KUKA KRL program: EPS_2_25694_GD06_A_20260114065907.src

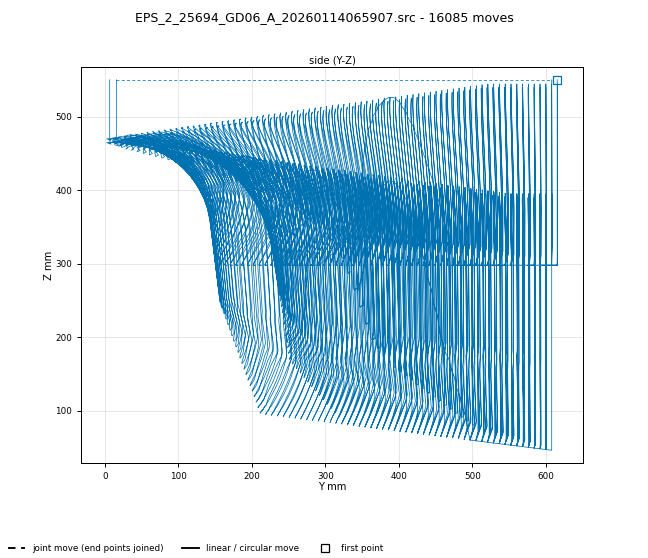
[picture p0: tool path of EPS_2_25694_GD06_A_20260114065907.src, 16085 of 16087 moves have a stored position in this frame; points joined in program order, loops and branches not executed]
&ACCESS RVP
&REL 4
&COMMENT QRS 19112012
&PARAM EDITMASK = *
DEF PART()
EXT BAS (BAS_COMMAND :IN,REAL :IN )
INT I
BAS (#INITMOV,0 )

;KUKA QRS Post kuka4.cps  Date:22-06-2017 !

File_ID=2966

QRS_PRE_INIT()

;Init var - Until changes are made in qrs_pre_init
Outlet_Square_prg=0
Inlet_1_Square_prg=0
Inlet_2_Square_prg=0
Inlet_3_Square_prg=0
Inlet_4_Square_prg=0
Inlet_5_Square_prg=0

Outlet_1={X 0.000, Y 524.050, Z 357.000, B 0.000, E1 0.000 }
Inlet_1={X 0.000, Y 548.960, Z 269.500, B 0.000, E1 174.000 }
Inlet_2={X 0.000, Y 548.960, Z 269.500, B 0.000, E1 220.000 }
Outlet_1_type=366
Inlet_1_type=201
Inlet_2_type=201
;QRS#1=Sidecore dimensions
;QRS#2=375-15" PVC SDR 35
;QRS#3=200-8" PVC SDR 35
;QRS#4=200-8" PVC SDR 35
;QRS#5=
;QRS#6=
;QRS#7=
;QRS#8=
;QRS#9=20Y PSX
;QRS#10=12-08 PSX
;QRS#11=12-08 PSX
;QRS#12=
;QRS#13=
;QRS#14=
;QRS#15=
;QRS#16=1220x127x838 2,75'
;QRS#17=EPS Height
;QRS#18=540
;QRS#19=*
;QRS#20= UPDATED VERSION 22-06-2017
;QRS#21=*
Outlet_Square=0250
Inlet_1_Square=0100
Inlet_2_Square=0100
Inlet_3_Square=0
Inlet_4_Square=0
Inlet_5_Square=0
Mill_Square=1
Outlet_Square_Prg=252
Inlet_1_Square_prg=204
Inlet_2_Square_prg=204

QRS_INIT()

$ADVANCE=5

; T1
PTP {E1 172.623,E2 172.623}
PTP {X 0,Y 615.402,A -85,B 0,C 180,E1 172.623,E2 172.623,E3 0,E4 0,E5 0,E6 0}
QRS_SPEED_INIT()
LIN {X 0,Y 615.402,Z 550,A -85,B 0,C 180,E1 172.623,E2 172.623,E3 0,E4 0,E5 0,E6 0} C_VEL
LIN {X 0,Y 615.402,Z 299.81,A -85,B 0,C 180,E1 172.623,E2 172.623} C_VEL
LIN {X 0,Y 615.427,Z 297.81,A -85,B 0,C 180,E1 172.809,E2 172.809} C_VEL
LIN {X 0,Y 615.817,Z 297.81,A -85,B 0,C 180,E1 174.193,E2 174.193} C_VEL
LIN {X 0,Y 615.867,Z 297.81,A -85,B 0,C 180,E1 178.841,E2 178.841} C_VEL
LIN {X 0,Y 615.867,Z 297.81,A -85,B 0,C 180,E1 183.48,E2 183.48} C_VEL
LIN {X 0,Y 615.824,Z 297.81,A -85,B 0,C 180,E1 188.143,E2 188.143} C_VEL
LIN {X 0,Y 615.832,Z 297.81,A -85,B 0,C 180,E1 192.861,E2 192.861} C_VEL
LIN {X 0,Y 615.792,Z 297.81,A -85,B 0,C 180,E1 197.671,E2 197.671} C_VEL
LIN {X 0,Y 615.792,Z 297.81,A -85,B 0,C 180,E1 197.997,E2 197.997} C_VEL
LIN {X 0,Y 615.78,Z 297.81,A -85,B 0,C 180,E1 202.613,E2 202.613} C_VEL
LIN {X 0,Y 615.256,Z 297.81,A -85,B 0,C 180,E1 205.172,E2 205.172} C_VEL
LIN {X 0,Y 615.748,Z 297.81,A -85,B 0,C 180,E1 207.741,E2 207.741} C_VEL
LIN {X 0,Y 615.184,Z 297.81,A -85,B 0,C 180,E1 210.425,E2 210.425} C_VEL
LIN {X 0,Y 615.704,Z 297.81,A -85,B 0,C 180,E1 213.124,E2 213.124} C_VEL
LIN {X 0,Y 615.631,Z 297.81,A -85,B 0,C 180,E1 213.914,E2 213.914} C_VEL
LIN {X 0,Y 615.66,Z 297.81,A -85,B 0,C 180,E1 218.863,E2 218.863} C_VEL
LIN {X 0,Y 615.262,Z 297.81,A -85,B 0,C 180,E1 221.942,E2 221.942} C_VEL
LIN {X 0,Y 615.675,Z 297.81,A -85,B 0,C 180,E1 224.897,E2 224.897} C_VEL
LIN {X 0,Y 615.638,Z 297.81,A -85,B 0,C 180,E1 228.498,E2 228.498} C_VEL
LIN {X 0,Y 615.376,Z 297.81,A -85,B 0,C 180,E1 231.118,E2 231.118} C_VEL
LIN {X 0,Y 615.432,Z 297.81,A -85,B 0,C 180,E1 232.156,E2 232.156} C_VEL
LIN {X 0,Y 615.702,Z 297.81,A -85,B 0,C 180,E1 234.062,E2 234.062} C_VEL
LIN {X 0,Y 615.153,Z 297.81,A -85,B 0,C 180,E1 236.844,E2 236.844} C_VEL
LIN {X 0,Y 615.737,Z 297.81,A -85,B 0,C 180,E1 239.607,E2 239.607} C_VEL
LIN {X 0,Y 615.234,Z 297.81,A -85,B 0,C 180,E1 242.236,E2 242.236} C_VEL
LIN {X 0,Y 615.794,Z 297.81,A -85,B 0,C 180,E1 244.853,E2 244.853} C_VEL
LIN {X 0,Y 615.734,Z 297.81,A -85,B 0,C 180,E1 247.988,E2 247.988} C_VEL
LIN {X 0,Y 615.838,Z 297.81,A -85,B 0,C 180,E1 248.694,E2 248.694} C_VEL
LIN {X 0,Y 615.498,Z 297.81,A -85,B 0,C 180,E1 249.163,E2 249.163} C_VEL
LIN {X 0,Y 615.621,Z 310.955,A -85,B 0,C 180,E1 249.342,E2 249.342} C_VEL
LIN {X 0,Y 615.725,Z 356.141,A -85,B 0,C 180,E1 249.896,E2 249.896} C_VEL
LIN {X 0,Y 615.805,Z 368.255,A -85,B 0,C 180,E1 250.073,E2 250.073} C_VEL
LIN {X 0,Y 615.746,Z 379.719,A -85,B 0,C 180,E1 250.302,E2 250.302} C_VEL
LIN {X 0,Y 615.701,Z 387.593,A -85,B 0,C 180,E1 250.493,E2 250.493} C_VEL
LIN {X 0,Y 615.787,Z 397.991,A -85,B 0,C 180,E1 250.803,E2 250.803} C_VEL
LIN {X 0,Y 615.773,Z 406.896,A -85,B 0,C 180,E1 251.109,E2 251.109} C_VEL
LIN {X 0,Y 615.749,Z 416.189,A -85,B 0,C 180,E1 251.476,E2 251.476} C_VEL
LIN {X 0,Y 615.792,Z 425.493,A -85,B 0,C 180,E1 251.897,E2 251.897} C_VEL
LIN {X 0,Y 615.792,Z 434.075,A -85,B 0,C 180,E1 252.331,E2 252.331} C_VEL
LIN {X 0,Y 615.784,Z 442.97,A -85,B 0,C 180,E1 252.832,E2 252.832} C_VEL
LIN {X 0,Y 615.789,Z 450.993,A -85,B 0,C 180,E1 253.333,E2 253.333} C_VEL
LIN {X 0,Y 615.781,Z 459.321,A -85,B 0,C 180,E1 253.906,E2 253.906} C_VEL
LIN {X 0,Y 615.8,Z 466.259,A -85,B 0,C 180,E1 254.428,E2 254.428} C_VEL
LIN {X 0,Y 615.798,Z 473.812,A -85,B 0,C 180,E1 255.049,E2 255.049} C_VEL
LIN {X 0,Y 615.765,Z 480.491,A -85,B 0,C 180,E1 255.648,E2 255.648} C_VEL
LIN {X 0,Y 615.798,Z 486.621,A -85,B 0,C 180,E1 256.246,E2 256.246} C_VEL
LIN {X 0,Y 615.819,Z 492.276,A -85,B 0,C 180,E1 256.842,E2 256.842} C_VEL
LIN {X 0,Y 615.737,Z 498.725,A -85,B 0,C 180,E1 257.584,E2 257.584} C_VEL
LIN {X 0,Y 615.725,Z 504.582,A -85,B 0,C 180,E1 258.325,E2 258.325} C_VEL
LIN {X 0,Y 615.783,Z 508.909,A -85,B 0,C 180,E1 258.917,E2 258.917} C_VEL
LIN {X 0,Y 615.79,Z 514.734,A -85,B 0,C 180,E1 259.802,E2 259.802} C_VEL
LIN {X 0,Y 615.671,Z 519.943,A -85,B 0,C 180,E1 260.683,E2 260.683} C_VEL
LIN {X 0,Y 615.681,Z 523.126,A -85,B 0,C 180,E1 261.27,E2 261.27} C_VEL
LIN {X 0,Y 615.809,Z 527.25,A -85,B 0,C 180,E1 262.129,E2 262.129} C_VEL
LIN {X 0,Y 615.715,Z 531.738,A -85,B 0,C 180,E1 263.207,E2 263.207} C_VEL
LIN {X 0,Y 615.679,Z 534.167,A -85,B 0,C 180,E1 263.864,E2 263.864} C_VEL
LIN {X 0,Y 615.737,Z 536.697,A -85,B 0,C 180,E1 264.659,E2 264.659} C_VEL
LIN {X 0,Y 615.8,Z 539.18,A -85,B 0,C 180,E1 265.591,E2 265.591} C_VEL
LIN {X 0,Y 615.655,Z 541.197,A -85,B 0,C 180,E1 266.52,E2 266.52} C_VEL
LIN {X 0,Y 615.667,Z 542.698,A -85,B 0,C 180,E1 267.449,E2 267.449} C_VEL
LIN {X 0,Y 615.73,Z 543.233,A -85,B 0,C 180,E1 267.913,E2 267.913} C_VEL
LIN {X 0,Y 615.79,Z 544.034,A -85,B 0,C 180,E1 268.841,E2 268.841} C_VEL
LIN {X 0,Y 615.643,Z 544.415,A -85,B 0,C 180,E1 269.769,E2 269.769} C_VEL
LIN {X 0,Y 615.659,Z 544.303,A -85,B 0,C 180,E1 270.697,E2 270.697} C_VEL
LIN {X 0,Y 615.728,Z 544.045,A -85,B 0,C 180,E1 271.16,E2 271.16} C_VEL
LIN {X 0,Y 615.709,Z 542.688,A -85,B 0,C 180,E1 272.553,E2 272.553} C_VEL
LIN {X 0,Y 615.632,Z 541.198,A -85,B 0,C 180,E1 273.482,E2 273.482} C_VEL
LIN {X 0,Y 615.743,Z 539.186,A -85,B 0,C 180,E1 274.411,E2 274.411} C_VEL
LIN {X 0,Y 615.793,Z 536.681,A -85,B 0,C 180,E1 275.342,E2 275.342} C_VEL
LIN {X 0,Y 615.685,Z 533.647,A -85,B 0,C 180,E1 276.284,E2 276.284} C_VEL
LIN {X 0,Y 615.732,Z 530.365,A -85,B 0,C 180,E1 277.148,E2 277.148} C_VEL
LIN {X 0,Y 615.811,Z 525.949,A -85,B 0,C 180,E1 278.144,E2 278.144} C_VEL
LIN {X 0,Y 615.693,Z 521.532,A -85,B 0,C 180,E1 279.025,E2 279.025} C_VEL
LIN {X 0,Y 615.673,Z 518.31,A -85,B 0,C 180,E1 279.613,E2 279.613} C_VEL
LIN {X 0,Y 615.794,Z 512.856,A -85,B 0,C 180,E1 280.494,E2 280.494} C_VEL
LIN {X 0,Y 615.803,Z 507.842,A -85,B 0,C 180,E1 281.232,E2 281.232} C_VEL
LIN {X 0,Y 615.711,Z 501.118,A -85,B 0,C 180,E1 282.122,E2 282.122} C_VEL
LIN {X 0,Y 615.758,Z 494.899,A -85,B 0,C 180,E1 282.863,E2 282.863} C_VEL
LIN {X 0,Y 615.835,Z 489.481,A -85,B 0,C 180,E1 283.457,E2 283.457} C_VEL
LIN {X 0,Y 615.797,Z 483.617,A -85,B 0,C 180,E1 284.054,E2 284.054} C_VEL
LIN {X 0,Y 615.767,Z 477.229,A -85,B 0,C 180,E1 284.654,E2 284.654} C_VEL
LIN {X 0,Y 615.775,Z 469.18,A -85,B 0,C 180,E1 285.339,E2 285.339} C_VEL
LIN {X 0,Y 615.798,Z 462.064,A -85,B 0,C 180,E1 285.893,E2 285.893} C_VEL
LIN {X 0,Y 615.802,Z 454.236,A -85,B 0,C 180,E1 286.45,E2 286.45} C_VEL
LIN {X 0,Y 615.788,Z 445.662,A -85,B 0,C 180,E1 287.005,E2 287.005} C_VEL
LIN {X 0,Y 615.783,Z 437.089,A -85,B 0,C 180,E1 287.505,E2 287.505} C_VEL
LIN {X 0,Y 615.774,Z 429.098,A -85,B 0,C 180,E1 287.926,E2 287.926} C_VEL
LIN {X 0,Y 615.807,Z 420.867,A -85,B 0,C 180,E1 288.317,E2 288.317} C_VEL
LIN {X 0,Y 615.769,Z 412.278,A -85,B 0,C 180,E1 288.684,E2 288.684} C_VEL
LIN {X 0,Y 615.728,Z 403.668,A -85,B 0,C 180,E1 289.009,E2 289.009} C_VEL
LIN {X 0,Y 615.82,Z 392.91,A -85,B 0,C 180,E1 289.352,E2 289.352} C_VEL
LIN {X 0,Y 615.806,Z 383.689,A -85,B 0,C 180,E1 289.602,E2 289.602} C_VEL
LIN {X 0,Y 615.724,Z 374.227,A -85,B 0,C 180,E1 289.816,E2 289.816} C_VEL
LIN {X 0,Y 615.718,Z 364.366,A -85,B 0,C 180,E1 289.99,E2 289.99} C_VEL
LIN {X 0,Y 615.684,Z 340.1,A -85,B 0,C 180,E1 290.3,E2 290.3} C_VEL
LIN {X 0,Y 615.604,Z 309.449,A -85,B 0,C 180,E1 290.677,E2 290.677} C_VEL
LIN {X 0,Y 615.662,Z 297.81,A -85,B 0,C 180,E1 290.924,E2 290.924} C_VEL
LIN {X 0,Y 615.846,Z 297.81,A -85,B 0,C 180,E1 291.275,E2 291.275} C_VEL
LIN {X 0,Y 615.834,Z 297.81,A -85,B 0,C 180,E1 292.611,E2 292.611} C_VEL
LIN {X 0,Y 615.254,Z 297.81,A -85,B 0,C 180,E1 295.172,E2 295.172} C_VEL
LIN {X 0,Y 615.755,Z 297.81,A -85,B 0,C 180,E1 297.741,E2 297.741} C_VEL
LIN {X 0,Y 615.188,Z 297.81,A -85,B 0,C 180,E1 300.425,E2 300.425} C_VEL
LIN {X 0,Y 615.704,Z 297.81,A -85,B 0,C 180,E1 303.125,E2 303.125} C_VEL
LIN {X 0,Y 615.639,Z 297.81,A -85,B 0,C 180,E1 303.912,E2 303.912} C_VEL
LIN {X 0,Y 615.631,Z 297.81,A -85,B 0,C 180,E1 308.865,E2 308.865} C_VEL
LIN {X 0,Y 615.208,Z 297.81,A -85,B 0,C 180,E1 311.946,E2 311.946} C_VEL
LIN {X 0,Y 615.608,Z 297.81,A -85,B 0,C 180,E1 314.888,E2 314.888} C_VEL
LIN {X 0,Y 615.621,Z 297.81,A -85,B 0,C 180,E1 318.5,E2 318.5} C_VEL
LIN {X 0,Y 615.341,Z 297.81,A -85,B 0,C 180,E1 321.113,E2 321.113} C_VEL
LIN {X 0,Y 615.391,Z 297.81,A -85,B 0,C 180,E1 322.16,E2 322.16} C_VEL
LIN {X 0,Y 615.638,Z 297.81,A -85,B 0,C 180,E1 324.056,E2 324.056} C_VEL
LIN {X 0,Y 615.107,Z 297.81,A -85,B 0,C 180,E1 326.839,E2 326.839} C_VEL
LIN {X 0,Y 615.705,Z 297.81,A -85,B 0,C 180,E1 329.604,E2 329.604} C_VEL
LIN {X 0,Y 615.204,Z 297.81,A -85,B 0,C 180,E1 332.233,E2 332.233} C_VEL
LIN {X 0,Y 615.747,Z 297.81,A -85,B 0,C 180,E1 334.85,E2 334.85} C_VEL
LIN {X 0,Y 615.745,Z 297.81,A -85,B 0,C 180,E1 339.877,E2 339.877} C_VEL
LIN {X 0,Y 615.773,Z 297.81,A -85,B 0,C 180,E1 343.783,E2 343.783} C_VEL
LIN {X 0,Y 615.771,Z 297.81,A -85,B 0,C 180,E1 349.506,E2 349.506} C_VEL
LIN {X 0,Y 615.834,Z 297.81,A -85,B 0,C 180,E1 354.193,E2 354.193} C_VEL
LIN {X 0,Y 615.858,Z 297.81,A -85,B 0,C 180,E1 358.841,E2 358.841} C_VEL
LIN {X 0,Y 615.81,Z 297.81,A -85,B 0,C 180,E1 363.48,E2 363.48} C_VEL
LIN {X 0,Y 615.85,Z 297.81,A -85,B 0,C 180,E1 368.143,E2 368.143} C_VEL
LIN {X 0,Y 615.774,Z 297.81,A -85,B 0,C 180,E1 372.862,E2 372.862} C_VEL
LIN {X 0,Y 615.794,Z 297.81,A -85,B 0,C 180,E1 377.671,E2 377.671} C_VEL
LIN {X 0,Y 615.796,Z 297.81,A -85,B 0,C 180,E1 377.992,E2 377.992} C_VEL
LIN {X 0,Y 615.745,Z 297.81,A -85,B 0,C 180,E1 382.614,E2 382.614} C_VEL
LIN {X 0,Y 615.221,Z 297.81,A -85,B 0,C 180,E1 385.173,E2 385.173} C_VEL
LIN {X 0,Y 615.747,Z 297.81,A -85,B 0,C 180,E1 387.741,E2 387.741} C_VEL
LIN {X 0,Y 615.229,Z 297.81,A -85,B 0,C 180,E1 390.422,E2 390.422} C_VEL
LIN {X 0,Y 615.823,Z 297.81,A -85,B 0,C 180,E1 393.117,E2 393.117} C_VEL
LIN {X 0,Y 615.838,Z 297.81,A -85,B 0,C 180,E1 397.92,E2 397.92} C_VEL
LIN {X 0,Y 615.79,Z 297.81,A -85,B 0,C 180,E1 398.066,E2 398.066} C_VEL
LIN {X 0,Y 615.611,Z 297.81,A -85,B 0,C 180,E1 398.128,E2 398.128} C_VEL
LIN {X 0,Y 615.791,Z 307.271,A -85,B 0,C 180,E1 398.409,E2 398.409} C_VEL
LIN {X 0,Y 615.852,Z 316.431,A -85,B 0,C 180,E1 398.75,E2 398.75} C_VEL
LIN {X 0,Y 615.848,Z 324.058,A -85,B 0,C 180,E1 399.093,E2 399.093} C_VEL
LIN {X 0,Y 615.861,Z 331.763,A -85,B 0,C 180,E1 399.5,E2 399.5} C_VEL
LIN {X 0,Y 615.839,Z 338.539,A -85,B 0,C 180,E1 399.916,E2 399.916} C_VEL
LIN {X 0,Y 615.815,Z 346.275,A -85,B 0,C 180,E1 400.463,E2 400.463} C_VEL
LIN {X 0,Y 615.85,Z 353.633,A -85,B 0,C 180,E1 401.07,E2 401.07} C_VEL
LIN {X 0,Y 615.809,Z 360.438,A -85,B 0,C 180,E1 401.723,E2 401.723} C_VEL
LIN {X 0,Y 615.772,Z 365.476,A -85,B 0,C 180,E1 402.271,E2 402.271} C_VEL
LIN {X 0,Y 615.81,Z 371.382,A -85,B 0,C 180,E1 403.019,E2 403.019} C_VEL
LIN {X 0,Y 615.813,Z 376.304,A -85,B 0,C 180,E1 403.741,E2 403.741} C_VEL
LIN {X 0,Y 615.749,Z 379.946,A -85,B 0,C 180,E1 404.36,E2 404.36} C_VEL
LIN {X 0,Y 615.79,Z 383.674,A -85,B 0,C 180,E1 405.095,E2 405.095} C_VEL
LIN {X 0,Y 615.832,Z 386.766,A -85,B 0,C 180,E1 405.836,E2 405.836} C_VEL
LIN {X 0,Y 615.744,Z 389.366,A -85,B 0,C 180,E1 406.585,E2 406.585} C_VEL
LIN {X 0,Y 615.764,Z 391.424,A -85,B 0,C 180,E1 407.348,E2 407.348} C_VEL
LIN {X 0,Y 615.84,Z 392.897,A -85,B 0,C 180,E1 408.106,E2 408.106} C_VEL
LIN {X 0,Y 615.797,Z 393.462,A -85,B 0,C 180,E1 408.481,E2 408.481} C_VEL
LIN {X 0,Y 615.766,Z 394.185,A -85,B 0,C 180,E1 409.228,E2 409.228} C_VEL
LIN {X 0,Y 615.803,Z 394.411,A -85,B 0,C 180,E1 409.833,E2 409.833} C_VEL
LIN {X 0,Y 615.843,Z 394.296,A -85,B 0,C 180,E1 410.496,E2 410.496} C_VEL
LIN {X 0,Y 615.768,Z 393.803,A -85,B 0,C 180,E1 411.145,E2 411.145} C_VEL
LIN {X 0,Y 615.795,Z 392.385,A -85,B 0,C 180,E1 412.112,E2 412.112} C_VEL
LIN {X 0,Y 615.822,Z 390.605,A -85,B 0,C 180,E1 412.881,E2 412.881} C_VEL
LIN {X 0,Y 615.73,Z 388.833,A -85,B 0,C 180,E1 413.492,E2 413.492} C_VEL
LIN {X 0,Y 615.742,Z 385.868,A -85,B 0,C 180,E1 414.312,E2 414.312} C_VEL
LIN {X 0,Y 615.829,Z 382.464,A -85,B 0,C 180,E1 415.062,E2 415.062} C_VEL
LIN {X 0,Y 615.787,Z 378.576,A -85,B 0,C 180,E1 415.797,E2 415.797} C_VEL
LIN {X 0,Y 615.8,Z 374.392,A -85,B 0,C 180,E1 416.462,E2 416.462} C_VEL
LIN {X 0,Y 615.851,Z 369.757,A -85,B 0,C 180,E1 417.108,E2 417.108} C_VEL
LIN {X 0,Y 615.805,Z 363.909,A -85,B 0,C 180,E1 417.813,E2 417.813} C_VEL
LIN {X 0,Y 615.811,Z 358.192,A -85,B 0,C 180,E1 418.416,E2 418.416} C_VEL
LIN {X 0,Y 615.849,Z 351.583,A -85,B 0,C 180,E1 419.016,E2 419.016} C_VEL
LIN {X 0,Y 615.82,Z 344.098,A -85,B 0,C 180,E1 419.609,E2 419.609} C_VEL
LIN {X 0,Y 615.835,Z 336.489,A -85,B 0,C 180,E1 420.127,E2 420.127} C_VEL
LIN {X 0,Y 615.822,Z 329.245,A -85,B 0,C 180,E1 420.55,E2 420.55} C_VEL
LIN {X 0,Y 615.826,Z 321.238,A -85,B 0,C 180,E1 420.952,E2 420.952} C_VEL
LIN {X 0,Y 615.807,Z 313.074,A -85,B 0,C 180,E1 421.295,E2 421.295} C_VEL
LIN {X 0,Y 615.702,Z 305.098,A -85,B 0,C 180,E1 421.573,E2 421.573} C_VEL
LIN {X 0,Y 615.384,Z 297.81,A -85,B 0,C 180,E1 421.796,E2 421.796} C_VEL
LIN {X 0,Y 615.784,Z 297.81,A -85,B 0,C 180,E1 421.916,E2 421.916} C_VEL
LIN {X 0,Y 615.706,Z 297.81,A -85,B 0,C 180,E1 423.559,E2 423.559} C_VEL
LIN {X 0,Y 615.767,Z 297.81,A -85,B 0,C 180,E1 424.85,E2 424.85} C_VEL
LIN {X 0,Y 615.813,Z 297.81,A -85,B 0,C 180,E1 429.878,E2 429.878} C_VEL
LIN {X 0,Y 615.83,Z 297.81,A -85,B 0,C 180,E1 433.784,E2 433.784} C_VEL
LIN {X 0,Y 615.806,Z 297.81,A -85,B 0,C 180,E1 439.506,E2 439.506} C_VEL
LIN {X 0,Y 615.79,Z 297.81,A -85,B 0,C 180,E1 443.78,E2 443.78} C_VEL
LIN {X 0,Y 615.666,Z 297.81,A -85,B 0,C 180,E1 443.985,E2 443.985} C_VEL
LIN {X 0,Y 615.253,Z 297.879,A -85,B 0,C 180,E1 444.123,E2 444.123} C_VEL
LIN {X 0,Y 615.743,Z 300.846,A -85,B 0,C 180,E1 444.213,E2 444.213} C_VEL
LIN {X 0,Y 615.794,Z 309.528,A -85,B 0,C 180,E1 444.483,E2 444.483} C_VEL
LIN {X 0,Y 615.801,Z 318.42,A -85,B 0,C 180,E1 444.833,E2 444.833} C_VEL
LIN {X 0,Y 615.828,Z 327,A -85,B 0,C 180,E1 445.24,E2 445.24} C_VEL
LIN {X 0,Y 615.826,Z 335.255,A -85,B 0,C 180,E1 445.705,E2 445.705} C_VEL
LIN {X 0,Y 615.823,Z 342.281,A -85,B 0,C 180,E1 446.17,E2 446.17} C_VEL
LIN {X 0,Y 615.804,Z 348.47,A -85,B 0,C 180,E1 446.635,E2 446.635} C_VEL
LIN {X 0,Y 615.834,Z 355.228,A -85,B 0,C 180,E1 447.216,E2 447.216} C_VEL
LIN {X 0,Y 615.856,Z 361.136,A -85,B 0,C 180,E1 447.796,E2 447.796} C_VEL
LIN {X 0,Y 615.795,Z 366.34,A -85,B 0,C 180,E1 448.376,E2 448.376} C_VEL
LIN {X 0,Y 615.812,Z 371.777,A -85,B 0,C 180,E1 449.072,E2 449.072} C_VEL
LIN {X 0,Y 615.857,Z 376.452,A -85,B 0,C 180,E1 449.767,E2 449.767} C_VEL
LIN {X 0,Y 615.782,Z 380.502,A -85,B 0,C 180,E1 450.463,E2 450.463} C_VEL
LIN {X 0,Y 615.758,Z 383.975,A -85,B 0,C 180,E1 451.159,E2 451.159} C_VEL
LIN {X 0,Y 615.804,Z 385.958,A -85,B 0,C 180,E1 451.623,E2 451.623} C_VEL
LIN {X 0,Y 615.855,Z 387.697,A -85,B 0,C 180,E1 452.086,E2 452.086} C_VEL
LIN {X 0,Y 615.803,Z 389.243,A -85,B 0,C 180,E1 452.551,E2 452.551} C_VEL
LIN {X 0,Y 615.766,Z 390.58,A -85,B 0,C 180,E1 453.015,E2 453.015} C_VEL
LIN {X 0,Y 615.756,Z 391.711,A -85,B 0,C 180,E1 453.48,E2 453.48} C_VEL
LIN {X 0,Y 615.843,Z 393.368,A -85,B 0,C 180,E1 454.409,E2 454.409} C_VEL
LIN {X 0,Y 615.784,Z 393.924,A -85,B 0,C 180,E1 454.875,E2 454.875} C_VEL
LIN {X 0,Y 615.721,Z 394.421,A -85,B 0,C 180,E1 455.807,E2 455.807} C_VEL
LIN {X 0,Y 615.746,Z 394.374,A -85,B 0,C 180,E1 456.281,E2 456.281} C_VEL
LIN {X 0,Y 615.812,Z 394.124,A -85,B 0,C 180,E1 456.756,E2 456.756} C_VEL
LIN {X 0,Y 615.781,Z 393.339,A -85,B 0,C 180,E1 457.535,E2 457.535} C_VEL
LIN {X 0,Y 615.722,Z 392.338,A -85,B 0,C 180,E1 458.143,E2 458.143} C_VEL
LIN {X 0,Y 615.73,Z 391.031,A -85,B 0,C 180,E1 458.73,E2 458.73} C_VEL
LIN {X 0,Y 615.85,Z 388.436,A -85,B 0,C 180,E1 459.609,E2 459.609} C_VEL
LIN {X 0,Y 615.793,Z 386.312,A -85,B 0,C 180,E1 460.198,E2 460.198} C_VEL
LIN {X 0,Y 615.747,Z 383.81,A -85,B 0,C 180,E1 460.788,E2 460.788} C_VEL
LIN {X 0,Y 615.797,Z 379.255,A -85,B 0,C 180,E1 461.674,E2 461.674} C_VEL
LIN {X 0,Y 615.818,Z 374.709,A -85,B 0,C 180,E1 462.415,E2 462.415} C_VEL
LIN {X 0,Y 615.776,Z 369.397,A -85,B 0,C 180,E1 463.158,E2 463.158} C_VEL
LIN {X 0,Y 615.815,Z 364.439,A -85,B 0,C 180,E1 463.754,E2 463.754} C_VEL
LIN {X 0,Y 615.846,Z 358.824,A -85,B 0,C 180,E1 464.351,E2 464.351} C_VEL
LIN {X 0,Y 615.804,Z 352.362,A -85,B 0,C 180,E1 464.951,E2 464.951} C_VEL
LIN {X 0,Y 615.817,Z 344.84,A -85,B 0,C 180,E1 465.556,E2 465.556} C_VEL
LIN {X 0,Y 615.823,Z 338.349,A -85,B 0,C 180,E1 466.006,E2 466.006} C_VEL
LIN {X 0,Y 615.832,Z 330.956,A -85,B 0,C 180,E1 466.458,E2 466.458} C_VEL
LIN {X 0,Y 615.844,Z 323.163,A -85,B 0,C 180,E1 466.86,E2 466.86} C_VEL
LIN {X 0,Y 615.843,Z 315.191,A -85,B 0,C 180,E1 467.213,E2 467.213} C_VEL
LIN {X 0,Y 615.838,Z 306.773,A -85,B 0,C 180,E1 467.516,E2 467.516} C_VEL
LIN {X 0,Y 615.737,Z 297.81,A -85,B 0,C 180,E1 467.787,E2 467.787} C_VEL
LIN {X 0,Y 615.787,Z 297.81,A -85,B 0,C 180,E1 470.121,E2 470.121} C_VEL
LIN {X 0,Y 615.755,Z 297.81,A -85,B 0,C 180,E1 475.148,E2 475.148} C_VEL
LIN {X 0,Y 615.416,Z 297.81,A -85,B 0,C 180,E1 479.461,E2 479.461} C_VEL
LIN {X 0,Y 615.746,Z 297.81,A -85,B 0,C 180,E1 480.393,E2 480.393} C_VEL
LIN {X 0,Y 615.157,Z 297.81,A -85,B 0,C 180,E1 483.845,E2 483.845} C_VEL
LIN {X 0,Y 615.692,Z 297.81,A -85,B 0,C 180,E1 485.939,E2 485.939} C_VEL
LIN {X 0,Y 615.645,Z 297.81,A -85,B 0,C 180,E1 487.87,E2 487.87} C_VEL
LIN {X 0,Y 615.726,Z 297.81,A -85,B 0,C 180,E1 488.856,E2 488.856} C_VEL
LIN {X 0,Y 615.226,Z 297.81,A -85,B 0,C 180,E1 491.943,E2 491.943} C_VEL
LIN {X 0,Y 615.649,Z 297.81,A -85,B 0,C 180,E1 494.892,E2 494.892} C_VEL
LIN {X 0,Y 615.618,Z 297.81,A -85,B 0,C 180,E1 498.498,E2 498.498} C_VEL
LIN {X 0,Y 615.356,Z 297.81,A -85,B 0,C 180,E1 501.114,E2 501.114} C_VEL
LIN {X 0,Y 615.409,Z 297.81,A -85,B 0,C 180,E1 502.155,E2 502.155} C_VEL
LIN {X 0,Y 615.689,Z 297.81,A -85,B 0,C 180,E1 504.059,E2 504.059} C_VEL
LIN {X 0,Y 615.136,Z 297.81,A -85,B 0,C 180,E1 506.841,E2 506.841} C_VEL
LIN {X 0,Y 615.715,Z 297.81,A -85,B 0,C 180,E1 509.604,E2 509.604} C_VEL
LIN {X 0,Y 615.204,Z 297.81,A -85,B 0,C 180,E1 512.233,E2 512.233} C_VEL
LIN {X 0,Y 615.732,Z 297.81,A -85,B 0,C 180,E1 514.849,E2 514.849} C_VEL
LIN {X 0,Y 615.817,Z 297.81,A -85,B 0,C 180,E1 519.879,E2 519.879} C_VEL
LIN {X 0,Y 615.772,Z 297.81,A -85,B 0,C 180,E1 523.3,E2 523.3} C_VEL
LIN {X 0,Y 615.423,Z 297.81,A -85,B 0,C 180,E1 524.738,E2 524.738} C_VEL
LIN {X 0,Y 615.844,Z 297.81,A -85,B 0,C 180,E1 529.507,E2 529.507} C_VEL
LIN {X 0,Y 615.427,Z 297.81,A -85,B 0,C 180,E1 532.809,E2 532.809} C_VEL
LIN {X 0,Y 612.995,Z 297.81,A -85,B 0,C 180,E1 534.011,E2 534.011} C_VEL
LIN {X 0,Y 607.578,Z 297.81,A -85,B 0,C 180,E1 535.808,E2 535.808} C_VEL
LIN {X 0,Y 607.469,Z 297.81,A -85,B 0,C 180,E1 536.015,E2 536.015} C_VEL
LIN {X 0,Y 607.617,Z 297.81,A -85,B 0,C 180,E1 539.991,E2 539.991} C_VEL
LIN {X 0,Y 607.701,Z 297.81,A -85,B 0,C 180,E1 544.263,E2 544.263} C_VEL
LIN {X 0,Y 607.775,Z 297.81,A -85,B 0,C 180,E1 548.558,E2 548.558} C_VEL
LIN {X 0,Y 607.925,Z 297.81,A -85,B 0,C 180,E1 552.9,E2 552.9} C_VEL
LIN {X 0,Y 607.621,Z 297.81,A -85,B 0,C 180,E1 558.827,E2 558.827} C_VEL
LIN {X 0,Y 607.588,Z 297.81,A -85,B 0,C 180,E1 563.405,E2 563.405} C_VEL
LIN {X 0,Y 607.693,Z 297.81,A -85,B 0,C 180,E1 568.142,E2 568.142} C_VEL
LIN {X 0,Y 607.805,Z 297.81,A -85,B 0,C 180,E1 573.097,E2 573.097} C_VEL
LIN {X 0,Y 607.509,Z 297.81,A -85,B 0,C 180,E1 579.645,E2 579.645} C_VEL
LIN {X 0,Y 607.535,Z 297.81,A -85,B 0,C 180,E1 585.935,E2 585.935} C_VEL
LIN {X 0,Y 607.438,Z 297.81,A -85,B 0,C 180,E1 590.351,E2 590.351} C_VEL
LIN {X 0,Y 607.429,Z 297.81,A -85,B 0,C 180,E1 595.153,E2 595.153} C_VEL
LIN {X 0,Y 607.58,Z 297.81,A -85,B 0,C 180,E1 600.359,E2 600.359} C_VEL
LIN {X 0,Y 607.866,Z 297.81,A -85,B 0,C 180,E1 605.038,E2 605.038} C_VEL
LIN {X 0,Y 607.771,Z 297.81,A -85,B 0,C 180,E1 608.899,E2 608.899} C_VEL
LIN {X 0,Y 608.338,Z 378.776,A -85,B 0,C 180,E1 610.029,E2 610.029} C_VEL
LIN {X 0,Y 608.256,Z 411.502,A -85,B 0,C 180,E1 611.046,E2 611.046} C_VEL
LIN {X 0,Y 608.14,Z 444.064,A -85,B 0,C 180,E1 612.676,E2 612.676} C_VEL
LIN {X 0,Y 608.084,Z 472.977,A -85,B 0,C 180,E1 614.78,E2 614.78} C_VEL
LIN {X 0,Y 607.951,Z 497.622,A -85,B 0,C 180,E1 617.274,E2 617.274} C_VEL
LIN {X 0,Y 607.898,Z 516.906,A -85,B 0,C 180,E1 619.993,E2 619.993} C_VEL
LIN {X 0,Y 607.876,Z 531.186,A -85,B 0,C 180,E1 622.87,E2 622.87} C_VEL
LIN {X 0,Y 607.892,Z 540.101,A -85,B 0,C 180,E1 625.729,E2 625.729} C_VEL
LIN {X 0,Y 607.881,Z 544.419,A -85,B 0,C 180,E1 628.577,E2 628.577} C_VEL
LIN {X 0,Y 607.823,Z 544.419,A -85,B 0,C 180,E1 631.422,E2 631.422} C_VEL
LIN {X 0,Y 607.841,Z 540.103,A -85,B 0,C 180,E1 634.271,E2 634.271} C_VEL
LIN {X 0,Y 607.891,Z 530.086,A -85,B 0,C 180,E1 637.39,E2 637.39} C_VEL
LIN {X 0,Y 607.931,Z 514.736,A -85,B 0,C 180,E1 640.367,E2 640.367} C_VEL
LIN {X 0,Y 607.969,Z 494.45,A -85,B 0,C 180,E1 643.09,E2 643.09} C_VEL
LIN {X 0,Y 608.069,Z 468.731,A -85,B 0,C 180,E1 645.575,E2 645.575} C_VEL
LIN {X 0,Y 608.18,Z 439.431,A -85,B 0,C 180,E1 647.601,E2 647.601} C_VEL
LIN {X 0,Y 608.251,Z 407.802,A -85,B 0,C 180,E1 649.098,E2 649.098} C_VEL
LIN {X 0,Y 608.289,Z 373.526,A -85,B 0,C 180,E1 650.082,E2 650.082} C_VEL
LIN {X 0,Y 607.842,Z 297.81,A -85,B 0,C 180,E1 651.098,E2 651.098} C_VEL
LIN {X 0,Y 607.511,Z 297.81,A -85,B 0,C 180,E1 656.61,E2 656.61} C_VEL
LIN {X 0,Y 607.539,Z 297.81,A -85,B 0,C 180,E1 662.397,E2 662.397} C_VEL
LIN {X 0,Y 607.552,Z 297.81,A -85,B 0,C 180,E1 668.384,E2 668.384} C_VEL
LIN {X 0,Y 607.449,Z 297.81,A -85,B 0,C 180,E1 674.071,E2 674.071} C_VEL
LIN {X 0,Y 607.633,Z 297.81,A -85,B 0,C 180,E1 678.16,E2 678.16} C_VEL
LIN {X 0,Y 607.6,Z 297.81,A -85,B 0,C 180,E1 683.422,E2 683.422} C_VEL
LIN {X 0,Y 607.529,Z 297.81,A -85,B 0,C 180,E1 690.381,E2 690.381} C_VEL
LIN {X 0,Y 607.778,Z 297.81,A -85,B 0,C 180,E1 695.043,E2 695.043} C_VEL
LIN {X 0,Y 607.542,Z 297.81,A -85,B 0,C 180,E1 701.171,E2 701.171} C_VEL
LIN {X 0,Y 607.203,Z 297.81,A -85,B 0,C 180,E1 705.619,E2 705.619} C_VEL
LIN {X 0,Y 607.7,Z 297.81,A -85,B 0,C 180,E1 709.999,E2 709.999} C_VEL
LIN {X 0,Y 607.904,Z 297.81,A -85,B 0,C 180,E1 714.31,E2 714.31} C_VEL
LIN {X 0,Y 607.565,Z 297.81,A -85,B 0,C 180,E1 720.009,E2 720.009} C_VEL
LIN {X 0,Y 607.627,Z 297.81,A -85,B 0,C 180,E1 724.282,E2 724.282} C_VEL
LIN {X 0,Y 607.793,Z 297.81,A -85,B 0,C 180,E1 728.576,E2 728.576} C_VEL
LIN {X 0,Y 607.843,Z 297.81,A -85,B 0,C 180,E1 732.92,E2 732.92} C_VEL
LIN {X 0,Y 607.584,Z 297.81,A -85,B 0,C 180,E1 738.846,E2 738.846} C_VEL
LIN {X 0,Y 607.548,Z 297.81,A -85,B 0,C 180,E1 743.426,E2 743.426} C_VEL
LIN {X 0,Y 607.686,Z 297.81,A -85,B 0,C 180,E1 748.163,E2 748.163} C_VEL
LIN {X 0,Y 607.917,Z 297.81,A -85,B 0,C 180,E1 753.111,E2 753.111} C_VEL
LIN {X 0,Y 607.881,Z 297.869,A -85,B 0,C 180,E1 757.977,E2 757.977} C_VEL
LIN {X 0,Y 608.09,Z 324.763,A -85,B 0,C 180,E1 758.983,E2 758.983} C_VEL
LIN {X 0,Y 608.018,Z 347.922,A -85,B 0,C 180,E1 760.458,E2 760.458} C_VEL
LIN {X 0,Y 607.935,Z 366.539,A -85,B 0,C 180,E1 762.267,E2 762.267} C_VEL
LIN {X 0,Y 607.906,Z 381.719,A -85,B 0,C 180,E1 764.541,E2 764.541} C_VEL
LIN {X 0,Y 607.886,Z 391.02,A -85,B 0,C 180,E1 766.949,E2 766.949} C_VEL
LIN {X 0,Y 607.964,Z 393.551,A -85,B 0,C 180,E1 768.141,E2 768.141} C_VEL
LIN {X 0,Y 607.974,Z 394.922,A -85,B 0,C 180,E1 770.318,E2 770.318} C_VEL
LIN {X 0,Y 607.928,Z 391.925,A -85,B 0,C 180,E1 772.606,E2 772.606} C_VEL
LIN {X 0,Y 607.97,Z 383.474,A -85,B 0,C 180,E1 775.01,E2 775.01} C_VEL
LIN {X 0,Y 608.016,Z 369.234,A -85,B 0,C 180,E1 777.311,E2 777.311} C_VEL
LIN {X 0,Y 608.021,Z 349.649,A -85,B 0,C 180,E1 779.315,E2 779.315} C_VEL
LIN {X 0,Y 608.079,Z 326.178,A -85,B 0,C 180,E1 780.856,E2 780.856} C_VEL
LIN {X 0,Y 607.76,Z 300.878,A -85,B 0,C 180,E1 781.853,E2 781.853} C_VEL
LIN {X 0,Y 607.701,Z 297.81,A -85,B 0,C 180,E1 781.959,E2 781.959} C_VEL
LIN {X 0,Y 607.358,Z 297.81,A -85,B 0,C 180,E1 786.577,E2 786.577} C_VEL
LIN {X 0,Y 607.609,Z 297.81,A -85,B 0,C 180,E1 791.165,E2 791.165} C_VEL
LIN {X 0,Y 607.265,Z 297.81,A -85,B 0,C 180,E1 795.612,E2 795.612} C_VEL
LIN {X 0,Y 607.753,Z 297.81,A -85,B 0,C 180,E1 799.991,E2 799.991} C_VEL
LIN {X 0,Y 607.541,Z 298.465,A -85,B 0,C 180,E1 803.986,E2 803.986} C_VEL
LIN {X 0,Y 608.071,Z 323.644,A -85,B 0,C 180,E1 804.928,E2 804.928} C_VEL
LIN {X 0,Y 608.007,Z 346.615,A -85,B 0,C 180,E1 806.354,E2 806.354} C_VEL
LIN {X 0,Y 607.976,Z 366.175,A -85,B 0,C 180,E1 808.223,E2 808.223} C_VEL
LIN {X 0,Y 607.95,Z 380.712,A -85,B 0,C 180,E1 810.356,E2 810.356} C_VEL
LIN {X 0,Y 607.923,Z 390.743,A -85,B 0,C 180,E1 812.846,E2 812.846} C_VEL
LIN {X 0,Y 607.956,Z 393.765,A -85,B 0,C 180,E1 814.271,E2 814.271} C_VEL
LIN {X 0,Y 607.945,Z 394.691,A -85,B 0,C 180,E1 816.765,E2 816.765} C_VEL
LIN {X 0,Y 607.944,Z 390.125,A -85,B 0,C 180,E1 819.285,E2 819.285} C_VEL
LIN {X 0,Y 607.934,Z 379.279,A -85,B 0,C 180,E1 821.817,E2 821.817} C_VEL
LIN {X 0,Y 608.007,Z 363.38,A -85,B 0,C 180,E1 824.004,E2 824.004} C_VEL
LIN {X 0,Y 608.03,Z 342.745,A -85,B 0,C 180,E1 825.843,E2 825.843} C_VEL
LIN {X 0,Y 608.086,Z 319.29,A -85,B 0,C 180,E1 827.186,E2 827.186} C_VEL
LIN {X 0,Y 607.801,Z 297.81,A -85,B 0,C 180,E1 827.987,E2 827.987} C_VEL
LIN {X 0,Y 607.348,Z 297.81,A -85,B 0,C 180,E1 831.882,E2 831.882} C_VEL
LIN {X 0,Y 607.796,Z 297.81,A -85,B 0,C 180,E1 834.965,E2 834.965} C_VEL
LIN {X 0,Y 607.618,Z 297.81,A -85,B 0,C 180,E1 839.782,E2 839.782} C_VEL
LIN {X 0,Y 607.722,Z 297.81,A -85,B 0,C 180,E1 846.579,E2 846.579} C_VEL
LIN {X 0,Y 607.309,Z 297.81,A -85,B 0,C 180,E1 851.79,E2 851.79} C_VEL
LIN {X 0,Y 607.475,Z 297.81,A -85,B 0,C 180,E1 856.086,E2 856.086} C_VEL
LIN {X 0,Y 607.403,Z 297.81,A -85,B 0,C 180,E1 860.368,E2 860.368} C_VEL
LIN {X 0,Y 607.42,Z 297.81,A -85,B 0,C 180,E1 865.141,E2 865.141} C_VEL
LIN {X 0,Y 607.532,Z 297.81,A -85,B 0,C 180,E1 870.382,E2 870.382} C_VEL
LIN {X 0,Y 607.764,Z 297.81,A -85,B 0,C 180,E1 875.023,E2 875.023} C_VEL
LIN {X 0,Y 607.657,Z 297.81,A -85,B 0,C 180,E1 881.156,E2 881.156} C_VEL
LIN {X 0,Y 607.26,Z 297.81,A -85,B 0,C 180,E1 885.726,E2 885.726} C_VEL
LIN {X 0,Y 607.769,Z 297.81,A -85,B 0,C 180,E1 889.982,E2 889.982} C_VEL
LIN {X 0,Y 607.876,Z 297.81,A -85,B 0,C 180,E1 894.292,E2 894.292} C_VEL
LIN {X 0,Y 607.469,Z 297.81,A -85,B 0,C 180,E1 896.015,E2 896.015} C_VEL
LIN {X 0,Y 603.675,Z 297.81,A -85,B 0,C 180,E1 897.627,E2 897.627} C_VEL
LIN {X 0,Y 599.793,Z 297.81,A -85,B 0,C 180,E1 899.26,E2 899.26} C_VEL
LIN {X 0,Y 599.797,Z 297.81,A -85,B 0,C 180,E1 904.32,E2 904.32} C_VEL
LIN {X 0,Y 599.833,Z 297.81,A -85,B 0,C 180,E1 908.673,E2 908.673} C_VEL
LIN {X 0,Y 599.942,Z 297.81,A -85,B 0,C 180,E1 913.075,E2 913.075} C_VEL
LIN {X 0,Y 599.663,Z 297.81,A -85,B 0,C 180,E1 919.086,E2 919.086} C_VEL
LIN {X 0,Y 599.599,Z 297.81,A -85,B 0,C 180,E1 923.736,E2 923.736} C_VEL
LIN {X 0,Y 599.668,Z 297.81,A -85,B 0,C 180,E1 928.553,E2 928.553} C_VEL
LIN {X 0,Y 599.668,Z 297.81,A -85,B 0,C 180,E1 933.859,E2 933.859} C_VEL
LIN {X 0,Y 599.635,Z 297.81,A -85,B 0,C 180,E1 938.976,E2 938.976} C_VEL
LIN {X 0,Y 599.542,Z 297.81,A -85,B 0,C 180,E1 945.191,E2 945.191} C_VEL
LIN {X 0,Y 599.548,Z 297.81,A -85,B 0,C 180,E1 951.007,E2 951.007} C_VEL
LIN {X 0,Y 599.582,Z 297.81,A -85,B 0,C 180,E1 954.63,E2 954.63} C_VEL
LIN {X 0,Y 599.63,Z 297.81,A -85,B 0,C 180,E1 959.78,E2 959.78} C_VEL
LIN {X 0,Y 599.923,Z 297.81,A -85,B 0,C 180,E1 964.875,E2 964.875} C_VEL
LIN {X 0,Y 599.909,Z 297.81,A -85,B 0,C 180,E1 968.596,E2 968.596} C_VEL
LIN {X 0,Y 600.902,Z 335.691,A -85,B 0,C 180,E1 969.122,E2 969.122} C_VEL
LIN {X 0,Y 600.874,Z 380.906,A -85,B 0,C 180,E1 969.822,E2 969.822} C_VEL
LIN {X 0,Y 600.73,Z 414.949,A -85,B 0,C 180,E1 970.94,E2 970.94} C_VEL
LIN {X 0,Y 600.534,Z 446.068,A -85,B 0,C 180,E1 972.575,E2 972.575} C_VEL
LIN {X 0,Y 600.348,Z 474.286,A -85,B 0,C 180,E1 974.697,E2 974.697} C_VEL
LIN {X 0,Y 600.112,Z 499.089,A -85,B 0,C 180,E1 977.289,E2 977.289} C_VEL
LIN {X 0,Y 600.024,Z 519.061,A -85,B 0,C 180,E1 980.226,E2 980.226} C_VEL
LIN {X 0,Y 599.944,Z 533.192,A -85,B 0,C 180,E1 983.32,E2 983.32} C_VEL
LIN {X 0,Y 599.923,Z 541.631,A -85,B 0,C 180,E1 986.394,E2 986.394} C_VEL
LIN {X 0,Y 599.977,Z 544.42,A -85,B 0,C 180,E1 988.558,E2 988.558} C_VEL
LIN {X 0,Y 599.92,Z 544.42,A -85,B 0,C 180,E1 991.441,E2 991.441} C_VEL
LIN {X 0,Y 599.966,Z 540.103,A -85,B 0,C 180,E1 994.327,E2 994.327} C_VEL
LIN {X 0,Y 600.007,Z 529.67,A -85,B 0,C 180,E1 997.587,E2 997.587} C_VEL
LIN {X 0,Y 600.071,Z 515.136,A -85,B 0,C 180,E1 1000.437,E2 1000.437} C_VEL
LIN {X 0,Y 600.189,Z 494.451,A -85,B 0,C 180,E1 1003.263,E2 1003.263} C_VEL
LIN {X 0,Y 600.362,Z 468.864,A -85,B 0,C 180,E1 1005.769,E2 1005.769} C_VEL
LIN {X 0,Y 600.589,Z 439.435,A -85,B 0,C 180,E1 1007.831,E2 1007.831} C_VEL
LIN {X 0,Y 600.726,Z 406.822,A -85,B 0,C 180,E1 1009.386,E2 1009.386} C_VEL
LIN {X 0,Y 600.876,Z 373.869,A -85,B 0,C 180,E1 1010.334,E2 1010.334} C_VEL
LIN {X 0,Y 599.975,Z 297.81,A -85,B 0,C 180,E1 1011.392,E2 1011.392} C_VEL
LIN {X 0,Y 599.737,Z 297.81,A -85,B 0,C 180,E1 1018.297,E2 1018.297} C_VEL
LIN {X 0,Y 599.666,Z 297.81,A -85,B 0,C 180,E1 1023.872,E2 1023.872} C_VEL
LIN {X 0,Y 599.575,Z 297.81,A -85,B 0,C 180,E1 1028.99,E2 1028.99} C_VEL
LIN {X 0,Y 599.483,Z 297.81,A -85,B 0,C 180,E1 1035.197,E2 1035.197} C_VEL
LIN {X 0,Y 599.505,Z 297.81,A -85,B 0,C 180,E1 1041.014,E2 1041.014} C_VEL
LIN {X 0,Y 599.522,Z 297.81,A -85,B 0,C 180,E1 1044.636,E2 1044.636} C_VEL
LIN {X 0,Y 599.592,Z 297.81,A -85,B 0,C 180,E1 1049.788,E2 1049.788} C_VEL
LIN {X 0,Y 599.837,Z 297.81,A -85,B 0,C 180,E1 1054.909,E2 1054.909} C_VEL
LIN {X 0,Y 599.693,Z 297.81,A -85,B 0,C 180,E1 1060.915,E2 1060.915} C_VEL
LIN {X 0,Y 599.343,Z 297.81,A -85,B 0,C 180,E1 1065.426,E2 1065.426} C_VEL
LIN {X 0,Y 599.76,Z 297.81,A -85,B 0,C 180,E1 1069.865,E2 1069.865} C_VEL
LIN {X 0,Y 599.999,Z 297.81,A -85,B 0,C 180,E1 1074.235,E2 1074.235} C_VEL
LIN {X 0,Y 599.664,Z 297.81,A -85,B 0,C 180,E1 1080.009,E2 1080.009} C_VEL
LIN {X 0,Y 599.71,Z 297.81,A -85,B 0,C 180,E1 1084.338,E2 1084.338} C_VEL
LIN {X 0,Y 599.845,Z 297.81,A -85,B 0,C 180,E1 1088.691,E2 1088.691} C_VEL
LIN {X 0,Y 599.868,Z 297.81,A -85,B 0,C 180,E1 1093.095,E2 1093.095} C_VEL
LIN {X 0,Y 599.837,Z 297.81,A -85,B 0,C 180,E1 1097.581,E2 1097.581} C_VEL
LIN {X 0,Y 599.565,Z 297.81,A -85,B 0,C 180,E1 1103.757,E2 1103.757} C_VEL
LIN {X 0,Y 599.658,Z 297.81,A -85,B 0,C 180,E1 1108.574,E2 1108.574} C_VEL
LIN {X 0,Y 599.756,Z 297.81,A -85,B 0,C 180,E1 1113.873,E2 1113.873} C_VEL
LIN {X 0,Y 600.005,Z 297.81,A -85,B 0,C 180,E1 1117.799,E2 1117.799} C_VEL
LIN {X 0,Y 600.314,Z 325.6,A -85,B 0,C 180,E1 1118.881,E2 1118.881} C_VEL
LIN {X 0,Y 600.197,Z 349.487,A -85,B 0,C 180,E1 1120.458,E2 1120.458} C_VEL
LIN {X 0,Y 600.078,Z 368.526,A -85,B 0,C 180,E1 1122.413,E2 1122.413} C_VEL
LIN {X 0,Y 600.033,Z 382.151,A -85,B 0,C 180,E1 1124.557,E2 1124.557} C_VEL
LIN {X 0,Y 599.982,Z 390.86,A -85,B 0,C 180,E1 1126.849,E2 1126.849} C_VEL
LIN {X 0,Y 599.994,Z 394.712,A -85,B 0,C 180,E1 1129.164,E2 1129.164} C_VEL
LIN {X 0,Y 599.997,Z 394.276,A -85,B 0,C 180,E1 1131.245,E2 1131.245} C_VEL
LIN {X 0,Y 599.978,Z 389.239,A -85,B 0,C 180,E1 1133.611,E2 1133.611} C_VEL
LIN {X 0,Y 600.065,Z 378.052,A -85,B 0,C 180,E1 1136.103,E2 1136.103} C_VEL
LIN {X 0,Y 600.125,Z 361.637,A -85,B 0,C 180,E1 1138.303,E2 1138.303} C_VEL
LIN {X 0,Y 600.233,Z 340.091,A -85,B 0,C 180,E1 1140.162,E2 1140.162} C_VEL
LIN {X 0,Y 600.314,Z 316.083,A -85,B 0,C 180,E1 1141.472,E2 1141.472} C_VEL
LIN {X 0,Y 599.963,Z 297.81,A -85,B 0,C 180,E1 1142.17,E2 1142.17} C_VEL
LIN {X 0,Y 599.516,Z 297.81,A -85,B 0,C 180,E1 1146.252,E2 1146.252} C_VEL
LIN {X 0,Y 599.766,Z 297.81,A -85,B 0,C 180,E1 1150.909,E2 1150.909} C_VEL
LIN {X 0,Y 599.404,Z 297.81,A -85,B 0,C 180,E1 1155.419,E2 1155.419} C_VEL
LIN {X 0,Y 599.811,Z 297.81,A -85,B 0,C 180,E1 1159.857,E2 1159.857} C_VEL
LIN {X 0,Y 599.728,Z 297.81,A -85,B 0,C 180,E1 1163.801,E2 1163.801} C_VEL
LIN {X 0,Y 600.305,Z 325.238,A -85,B 0,C 180,E1 1164.863,E2 1164.863} C_VEL
LIN {X 0,Y 600.168,Z 348.727,A -85,B 0,C 180,E1 1166.397,E2 1166.397} C_VEL
LIN {X 0,Y 600.099,Z 368.261,A -85,B 0,C 180,E1 1168.379,E2 1168.379} C_VEL
LIN {X 0,Y 600.069,Z 381.137,A -85,B 0,C 180,E1 1170.361,E2 1170.361} C_VEL
LIN {X 0,Y 600.033,Z 390.951,A -85,B 0,C 180,E1 1172.883,E2 1172.883} C_VEL
LIN {X 0,Y 600.072,Z 393.88,A -85,B 0,C 180,E1 1174.327,E2 1174.327} C_VEL
LIN {X 0,Y 599.954,Z 394.966,A -85,B 0,C 180,E1 1175.775,E2 1175.775} C_VEL
LIN {X 0,Y 599.98,Z 393.29,A -85,B 0,C 180,E1 1177.952,E2 1177.952} C_VEL
LIN {X 0,Y 600.032,Z 386.433,A -85,B 0,C 180,E1 1180.399,E2 1180.399} C_VEL
LIN {X 0,Y 600.103,Z 374.232,A -85,B 0,C 180,E1 1182.711,E2 1182.711} C_VEL
LIN {X 0,Y 600.18,Z 356.545,A -85,B 0,C 180,E1 1184.819,E2 1184.819} C_VEL
LIN {X 0,Y 600.248,Z 335.285,A -85,B 0,C 180,E1 1186.478,E2 1186.478} C_VEL
LIN {X 0,Y 600.356,Z 310.343,A -85,B 0,C 180,E1 1187.697,E2 1187.697} C_VEL
LIN {X 0,Y 599.907,Z 297.81,A -85,B 0,C 180,E1 1188.137,E2 1188.137} C_VEL
LIN {X 0,Y 599.503,Z 297.81,A -85,B 0,C 180,E1 1193.75,E2 1193.75} C_VEL
LIN {X 0,Y 599.415,Z 297.81,A -85,B 0,C 180,E1 1198.576,E2 1198.576} C_VEL
LIN {X 0,Y 599.35,Z 297.81,A -85,B 0,C 180,E1 1203.795,E2 1203.795} C_VEL
LIN {X 0,Y 599.814,Z 297.81,A -85,B 0,C 180,E1 1208.733,E2 1208.733} C_VEL
LIN {X 0,Y 599.512,Z 297.81,A -85,B 0,C 180,E1 1215.174,E2 1215.174} C_VEL
LIN {X 0,Y 599.527,Z 297.81,A -85,B 0,C 180,E1 1220.993,E2 1220.993} C_VEL
LIN {X 0,Y 599.555,Z 297.81,A -85,B 0,C 180,E1 1224.616,E2 1224.616} C_VEL
LIN {X 0,Y 599.599,Z 297.81,A -85,B 0,C 180,E1 1229.768,E2 1229.768} C_VEL
LIN {X 0,Y 599.83,Z 297.81,A -85,B 0,C 180,E1 1234.912,E2 1234.912} C_VEL
LIN {X 0,Y 599.797,Z 297.81,A -85,B 0,C 180,E1 1240.899,E2 1240.899} C_VEL
LIN {X 0,Y 599.423,Z 297.81,A -85,B 0,C 180,E1 1245.41,E2 1245.41} C_VEL
LIN {X 0,Y 599.826,Z 297.81,A -85,B 0,C 180,E1 1249.848,E2 1249.848} C_VEL
LIN {X 0,Y 599.979,Z 297.81,A -85,B 0,C 180,E1 1254.217,E2 1254.217} C_VEL
LIN {X 0,Y 599.793,Z 297.81,A -85,B 0,C 180,E1 1259.26,E2 1259.26} C_VEL
LIN {X 0,Y 595.645,Z 297.81,A -85,B 0,C 180,E1 1260.891,E2 1260.891} C_VEL
LIN {X 0,Y 591.835,Z 297.81,A -85,B 0,C 180,E1 1262.544,E2 1262.544} C_VEL
LIN {X 0,Y 591.893,Z 297.81,A -85,B 0,C 180,E1 1268.79,E2 1268.79} C_VEL
LIN {X 0,Y 591.684,Z 297.81,A -85,B 0,C 180,E1 1274.272,E2 1274.272} C_VEL
LIN {X 0,Y 591.724,Z 297.81,A -85,B 0,C 180,E1 1279.352,E2 1279.352} C_VEL
LIN {X 0,Y 591.631,Z 297.81,A -85,B 0,C 180,E1 1284.076,E2 1284.076} C_VEL
LIN {X 0,Y 591.643,Z 297.81,A -85,B 0,C 180,E1 1288.977,E2 1288.977} C_VEL
LIN {X 0,Y 591.719,Z 297.81,A -85,B 0,C 180,E1 1294.118,E2 1294.118} C_VEL
LIN {X 0,Y 591.542,Z 297.81,A -85,B 0,C 180,E1 1300.067,E2 1300.067} C_VEL
LIN {X 0,Y 591.605,Z 297.81,A -85,B 0,C 180,E1 1305.566,E2 1305.566} C_VEL
LIN {X 0,Y 591.589,Z 297.81,A -85,B 0,C 180,E1 1310.38,E2 1310.38} C_VEL
LIN {X 0,Y 591.497,Z 297.81,A -85,B 0,C 180,E1 1315.857,E2 1315.857} C_VEL
LIN {X 0,Y 591.567,Z 297.81,A -85,B 0,C 180,E1 1321.009,E2 1321.009} C_VEL
LIN {X 0,Y 591.867,Z 297.81,A -85,B 0,C 180,E1 1326.594,E2 1326.594} C_VEL
LIN {X 0,Y 592,Z 297.81,A -85,B 0,C 180,E1 1328.295,E2 1328.295} C_VEL
LIN {X 0,Y 593.528,Z 312.319,A -85,B 0,C 180,E1 1328.553,E2 1328.553} C_VEL
LIN {X 0,Y 593.51,Z 378.641,A -85,B 0,C 180,E1 1329.505,E2 1329.505} C_VEL
LIN {X 0,Y 593.225,Z 411.48,A -85,B 0,C 180,E1 1330.546,E2 1330.546} C_VEL
LIN {X 0,Y 592.925,Z 444.072,A -85,B 0,C 180,E1 1332.217,E2 1332.217} C_VEL
LIN {X 0,Y 592.604,Z 473.242,A -85,B 0,C 180,E1 1334.397,E2 1334.397} C_VEL
LIN {X 0,Y 592.345,Z 497.624,A -85,B 0,C 180,E1 1336.933,E2 1336.933} C_VEL
LIN {X 0,Y 592.176,Z 517.993,A -85,B 0,C 180,E1 1339.91,E2 1339.91} C_VEL
LIN {X 0,Y 592.079,Z 532.289,A -85,B 0,C 180,E1 1342.981,E2 1342.981} C_VEL
LIN {X 0,Y 592.105,Z 540.102,A -85,B 0,C 180,E1 1345.615,E2 1345.615} C_VEL
LIN {X 0,Y 592.073,Z 544.42,A -85,B 0,C 180,E1 1348.539,E2 1348.539} C_VEL
LIN {X 0,Y 592.018,Z 544.421,A -85,B 0,C 180,E1 1351.46,E2 1351.46} C_VEL
LIN {X 0,Y 592.066,Z 540.104,A -85,B 0,C 180,E1 1354.385,E2 1354.385} C_VEL
LIN {X 0,Y 592.151,Z 529.67,A -85,B 0,C 180,E1 1357.688,E2 1357.688} C_VEL
LIN {X 0,Y 592.232,Z 513.781,A -85,B 0,C 180,E1 1360.803,E2 1360.803} C_VEL
LIN {X 0,Y 592.443,Z 493.173,A -85,B 0,C 180,E1 1363.589,E2 1363.589} C_VEL
LIN {X 0,Y 592.662,Z 467.729,A -85,B 0,C 180,E1 1366.074,E2 1366.074} C_VEL
LIN {X 0,Y 593.005,Z 437.758,A -85,B 0,C 180,E1 1368.163,E2 1368.163} C_VEL
LIN {X 0,Y 593.256,Z 406.292,A -85,B 0,C 180,E1 1369.661,E2 1369.661} C_VEL
LIN {X 0,Y 593.497,Z 372.089,A -85,B 0,C 180,E1 1370.634,E2 1370.634} C_VEL
LIN {X 0,Y 592.843,Z 301.233,A -85,B 0,C 180,E1 1371.614,E2 1371.614} C_VEL
LIN {X 0,Y 592.055,Z 297.81,A -85,B 0,C 180,E1 1371.721,E2 1371.721} C_VEL
LIN {X 0,Y 591.737,Z 297.81,A -85,B 0,C 180,E1 1377.323,E2 1377.323} C_VEL
LIN {X 0,Y 591.715,Z 297.81,A -85,B 0,C 180,E1 1384.128,E2 1384.128} C_VEL
LIN {X 0,Y 591.5,Z 297.81,A -85,B 0,C 180,E1 1390.075,E2 1390.075} C_VEL
LIN {X 0,Y 591.546,Z 297.81,A -85,B 0,C 180,E1 1395.582,E2 1395.582} C_VEL
LIN {X 0,Y 591.549,Z 297.81,A -85,B 0,C 180,E1 1400.387,E2 1400.387} C_VEL
LIN {X 0,Y 591.45,Z 297.81,A -85,B 0,C 180,E1 1405.864,E2 1405.864} C_VEL
LIN {X 0,Y 591.545,Z 297.81,A -85,B 0,C 180,E1 1411.018,E2 1411.018} C_VEL
LIN {X 0,Y 591.643,Z 297.81,A -85,B 0,C 180,E1 1415.925,E2 1415.925} C_VEL
LIN {X 0,Y 591.777,Z 297.81,A -85,B 0,C 180,E1 1420.65,E2 1420.65} C_VEL
LIN {X 0,Y 591.481,Z 297.81,A -85,B 0,C 180,E1 1425.228,E2 1425.228} C_VEL
LIN {X 0,Y 591.833,Z 297.81,A -85,B 0,C 180,E1 1429.728,E2 1429.728} C_VEL
LIN {X 0,Y 592.062,Z 297.81,A -85,B 0,C 180,E1 1434.158,E2 1434.158} C_VEL
LIN {X 0,Y 591.764,Z 297.81,A -85,B 0,C 180,E1 1440.009,E2 1440.009} C_VEL
LIN {X 0,Y 591.794,Z 297.81,A -85,B 0,C 180,E1 1444.396,E2 1444.396} C_VEL
LIN {X 0,Y 591.901,Z 297.81,A -85,B 0,C 180,E1 1448.808,E2 1448.808} C_VEL
LIN {X 0,Y 591.661,Z 297.81,A -85,B 0,C 180,E1 1454.267,E2 1454.267} C_VEL
LIN {X 0,Y 591.696,Z 297.81,A -85,B 0,C 180,E1 1459.372,E2 1459.372} C_VEL
LIN {X 0,Y 591.614,Z 297.81,A -85,B 0,C 180,E1 1464.097,E2 1464.097} C_VEL
LIN {X 0,Y 591.644,Z 297.81,A -85,B 0,C 180,E1 1468.998,E2 1468.998} C_VEL
LIN {X 0,Y 591.813,Z 297.81,A -85,B 0,C 180,E1 1474.134,E2 1474.134} C_VEL
LIN {X 0,Y 592.08,Z 298.561,A -85,B 0,C 180,E1 1477.671,E2 1477.671} C_VEL
LIN {X 0,Y 592.581,Z 324.166,A -85,B 0,C 180,E1 1478.662,E2 1478.662} C_VEL
LIN {X 0,Y 592.345,Z 347.389,A -85,B 0,C 180,E1 1480.161,E2 1480.161} C_VEL
LIN {X 0,Y 592.221,Z 367.2,A -85,B 0,C 180,E1 1482.144,E2 1482.144} C_VEL
LIN {X 0,Y 592.15,Z 382.116,A -85,B 0,C 180,E1 1484.477,E2 1484.477} C_VEL
LIN {X 0,Y 592.109,Z 391.68,A -85,B 0,C 180,E1 1487.124,E2 1487.124} C_VEL
LIN {X 0,Y 592.119,Z 394.11,A -85,B 0,C 180,E1 1488.502,E2 1488.502} C_VEL
LIN {X 0,Y 592.041,Z 394.901,A -85,B 0,C 180,E1 1490.417,E2 1490.417} C_VEL
LIN {X 0,Y 592.125,Z 391,A -85,B 0,C 180,E1 1493.049,E2 1493.049} C_VEL
LIN {X 0,Y 592.171,Z 381.324,A -85,B 0,C 180,E1 1495.588,E2 1495.588} C_VEL
LIN {X 0,Y 592.263,Z 366.664,A -85,B 0,C 180,E1 1497.832,E2 1497.832} C_VEL
LIN {X 0,Y 592.385,Z 346.333,A -85,B 0,C 180,E1 1499.834,E2 1499.834} C_VEL
LIN {X 0,Y 592.519,Z 323.038,A -85,B 0,C 180,E1 1501.305,E2 1501.305} C_VEL
LIN {X 0,Y 592.077,Z 297.81,A -85,B 0,C 180,E1 1502.278,E2 1502.278} C_VEL
LIN {X 0,Y 591.532,Z 297.81,A -85,B 0,C 180,E1 1507.503,E2 1507.503} C_VEL
LIN {X 0,Y 591.818,Z 297.81,A -85,B 0,C 180,E1 1512.184,E2 1512.184} C_VEL
LIN {X 0,Y 591.602,Z 297.81,A -85,B 0,C 180,E1 1518.226,E2 1518.226} C_VEL
LIN {X 0,Y 591.896,Z 297.81,A -85,B 0,C 180,E1 1523.645,E2 1523.645} C_VEL
LIN {X 0,Y 592.523,Z 323.186,A -85,B 0,C 180,E1 1524.612,E2 1524.612} C_VEL
LIN {X 0,Y 592.372,Z 346.338,A -85,B 0,C 180,E1 1526.075,E2 1526.075} C_VEL
LIN {X 0,Y 592.289,Z 365.975,A -85,B 0,C 180,E1 1527.993,E2 1527.993} C_VEL
LIN {X 0,Y 592.192,Z 381.549,A -85,B 0,C 180,E1 1530.365,E2 1530.365} C_VEL
LIN {X 0,Y 592.133,Z 391.158,A -85,B 0,C 180,E1 1532.922,E2 1532.922} C_VEL
LIN {X 0,Y 592.16,Z 393.974,A -85,B 0,C 180,E1 1534.385,E2 1534.385} C_VEL
LIN {X 0,Y 592.037,Z 394.961,A -85,B 0,C 180,E1 1536.157,E2 1536.157} C_VEL
LIN {X 0,Y 592.074,Z 391.652,A -85,B 0,C 180,E1 1538.797,E2 1538.797} C_VEL
LIN {X 0,Y 592.112,Z 383.241,A -85,B 0,C 180,E1 1541.196,E2 1541.196} C_VEL
LIN {X 0,Y 592.211,Z 368.814,A -85,B 0,C 180,E1 1543.562,E2 1543.562} C_VEL
LIN {X 0,Y 592.348,Z 349.102,A -85,B 0,C 180,E1 1545.61,E2 1545.61} C_VEL
LIN {X 0,Y 592.531,Z 325.963,A -85,B 0,C 180,E1 1547.157,E2 1547.157} C_VEL
LIN {X 0,Y 592.188,Z 299.413,A -85,B 0,C 180,E1 1548.213,E2 1548.213} C_VEL
LIN {X 0,Y 591.982,Z 297.81,A -85,B 0,C 180,E1 1548.388,E2 1548.388} C_VEL
LIN {X 0,Y 591.669,Z 297.81,A -85,B 0,C 180,E1 1554.084,E2 1554.084} C_VEL
LIN {X 0,Y 591.63,Z 297.81,A -85,B 0,C 180,E1 1559.844,E2 1559.844} C_VEL
LIN {X 0,Y 591.767,Z 297.81,A -85,B 0,C 180,E1 1565.909,E2 1565.909} C_VEL
LIN {X 0,Y 591.596,Z 297.81,A -85,B 0,C 180,E1 1570.057,E2 1570.057} C_VEL
LIN {X 0,Y 591.575,Z 297.81,A -85,B 0,C 180,E1 1575.58,E2 1575.58} C_VEL
LIN {X 0,Y 591.572,Z 297.81,A -85,B 0,C 180,E1 1580.366,E2 1580.366} C_VEL
LIN {X 0,Y 591.642,Z 297.81,A -85,B 0,C 180,E1 1584.704,E2 1584.704} C_VEL
LIN {X 0,Y 591.556,Z 297.81,A -85,B 0,C 180,E1 1590.998,E2 1590.998} C_VEL
LIN {X 0,Y 591.659,Z 297.81,A -85,B 0,C 180,E1 1595.905,E2 1595.905} C_VEL
LIN {X 0,Y 591.875,Z 297.81,A -85,B 0,C 180,E1 1600.634,E2 1600.634} C_VEL
LIN {X 0,Y 591.476,Z 297.81,A -85,B 0,C 180,E1 1605.807,E2 1605.807} C_VEL
LIN {X 0,Y 591.678,Z 297.81,A -85,B 0,C 180,E1 1611.188,E2 1611.188} C_VEL
LIN {X 0,Y 591.718,Z 297.81,A -85,B 0,C 180,E1 1615.603,E2 1615.603} C_VEL
LIN {X 0,Y 591.815,Z 297.81,A -85,B 0,C 180,E1 1619.991,E2 1619.991} C_VEL
LIN {X 0,Y 591.835,Z 297.81,A -85,B 0,C 180,E1 1622.544,E2 1622.544} C_VEL
LIN {X 0,Y 589.399,Z 297.81,A -85,B 0,C 180,E1 1623.794,E2 1623.794} C_VEL
LIN {X 0,Y 583.891,Z 297.81,A -85,B 0,C 180,E1 1625.663,E2 1625.663} C_VEL
LIN {X 0,Y 583.795,Z 297.81,A -85,B 0,C 180,E1 1625.879,E2 1625.879} C_VEL
LIN {X 0,Y 583.753,Z 297.81,A -85,B 0,C 180,E1 1630.795,E2 1630.795} C_VEL
LIN {X 0,Y 583.702,Z 297.81,A -85,B 0,C 180,E1 1634.973,E2 1634.973} C_VEL
LIN {X 0,Y 583.781,Z 297.81,A -85,B 0,C 180,E1 1639.626,E2 1639.626} C_VEL
LIN {X 0,Y 583.678,Z 297.81,A -85,B 0,C 180,E1 1644.425,E2 1644.425} C_VEL
LIN {X 0,Y 583.651,Z 297.81,A -85,B 0,C 180,E1 1649.412,E2 1649.412} C_VEL
LIN {X 0,Y 583.717,Z 297.81,A -85,B 0,C 180,E1 1654.652,E2 1654.652} C_VEL
LIN {X 0,Y 583.609,Z 297.81,A -85,B 0,C 180,E1 1660.261,E2 1660.261} C_VEL
LIN {X 0,Y 583.749,Z 297.81,A -85,B 0,C 180,E1 1666.358,E2 1666.358} C_VEL
LIN {X 0,Y 583.729,Z 297.81,A -85,B 0,C 180,E1 1671.652,E2 1671.652} C_VEL
LIN {X 0,Y 583.571,Z 297.81,A -85,B 0,C 180,E1 1677.11,E2 1677.11} C_VEL
LIN {X 0,Y 583.626,Z 297.81,A -85,B 0,C 180,E1 1682.263,E2 1682.263} C_VEL
LIN {X 0,Y 584.064,Z 297.81,A -85,B 0,C 180,E1 1687.824,E2 1687.824} C_VEL
LIN {X 0,Y 584.073,Z 297.81,A -85,B 0,C 180,E1 1687.989,E2 1687.989} C_VEL
LIN {X 0,Y 586.143,Z 308.497,A -85,B 0,C 180,E1 1688.22,E2 1688.22} C_VEL
LIN {X 0,Y 586.13,Z 377.575,A -85,B 0,C 180,E1 1689.208,E2 1689.208} C_VEL
LIN {X 0,Y 585.754,Z 411.484,A -85,B 0,C 180,E1 1690.287,E2 1690.287} C_VEL
LIN {X 0,Y 585.341,Z 444.076,A -85,B 0,C 180,E1 1691.979,E2 1691.979} C_VEL
LIN {X 0,Y 584.89,Z 473.241,A -85,B 0,C 180,E1 1694.186,E2 1694.186} C_VEL
LIN {X 0,Y 584.577,Z 497.624,A -85,B 0,C 180,E1 1696.756,E2 1696.756} C_VEL
LIN {X 0,Y 584.321,Z 517.993,A -85,B 0,C 180,E1 1699.773,E2 1699.773} C_VEL
LIN {X 0,Y 584.226,Z 531.185,A -85,B 0,C 180,E1 1702.579,E2 1702.579} C_VEL
LIN {X 0,Y 584.202,Z 540.102,A -85,B 0,C 180,E1 1705.555,E2 1705.555} C_VEL
LIN {X 0,Y 584.182,Z 544.421,A -85,B 0,C 180,E1 1708.519,E2 1708.519} C_VEL
LIN {X 0,Y 584.132,Z 544.421,A -85,B 0,C 180,E1 1711.48,E2 1711.48} C_VEL
LIN {X 0,Y 584.17,Z 540.103,A -85,B 0,C 180,E1 1714.444,E2 1714.444} C_VEL
LIN {X 0,Y 584.277,Z 529.67,A -85,B 0,C 180,E1 1717.792,E2 1717.792} C_VEL
LIN {X 0,Y 584.411,Z 513.379,A -85,B 0,C 180,E1 1721.012,E2 1721.012} C_VEL
LIN {X 0,Y 584.673,Z 492.213,A -85,B 0,C 180,E1 1723.888,E2 1723.888} C_VEL
LIN {X 0,Y 584.99,Z 466.588,A -85,B 0,C 180,E1 1726.387,E2 1726.387} C_VEL
LIN {X 0,Y 585.445,Z 437.762,A -85,B 0,C 180,E1 1728.405,E2 1728.405} C_VEL
LIN {X 0,Y 585.788,Z 406.289,A -85,B 0,C 180,E1 1729.922,E2 1729.922} C_VEL
LIN {X 0,Y 586.1,Z 372.899,A -85,B 0,C 180,E1 1730.89,E2 1730.89} C_VEL
LIN {X 0,Y 585.354,Z 302.617,A -85,B 0,C 180,E1 1731.887,E2 1731.887} C_VEL
LIN {X 0,Y 584.094,Z 297.81,A -85,B 0,C 180,E1 1732.078,E2 1732.078} C_VEL
LIN {X 0,Y 583.717,Z 297.81,A -85,B 0,C 180,E1 1738.5,E2 1738.5} C_VEL
LIN {X 0,Y 583.709,Z 297.81,A -85,B 0,C 180,E1 1744.662,E2 1744.662} C_VEL
LIN {X 0,Y 583.566,Z 297.81,A -85,B 0,C 180,E1 1750.274,E2 1750.274} C_VEL
LIN {X 0,Y 583.677,Z 297.81,A -85,B 0,C 180,E1 1756.376,E2 1756.376} C_VEL
LIN {X 0,Y 583.671,Z 297.81,A -85,B 0,C 180,E1 1761.659,E2 1761.659} C_VEL
LIN {X 0,Y 583.521,Z 297.81,A -85,B 0,C 180,E1 1767.117,E2 1767.117} C_VEL
LIN {X 0,Y 583.608,Z 297.81,A -85,B 0,C 180,E1 1772.272,E2 1772.272} C_VEL
LIN {X 0,Y 583.589,Z 297.81,A -85,B 0,C 180,E1 1777.188,E2 1777.188} C_VEL
LIN {X 0,Y 583.843,Z 297.81,A -85,B 0,C 180,E1 1781.941,E2 1781.941} C_VEL
LIN {X 0,Y 583.656,Z 297.81,A -85,B 0,C 180,E1 1788.072,E2 1788.072} C_VEL
LIN {X 0,Y 584.142,Z 297.81,A -85,B 0,C 180,E1 1794.078,E2 1794.078} C_VEL
LIN {X 0,Y 583.886,Z 297.81,A -85,B 0,C 180,E1 1800.009,E2 1800.009} C_VEL
LIN {X 0,Y 583.898,Z 297.81,A -85,B 0,C 180,E1 1804.456,E2 1804.456} C_VEL
LIN {X 0,Y 583.961,Z 297.81,A -85,B 0,C 180,E1 1808.929,E2 1808.929} C_VEL
LIN {X 0,Y 583.966,Z 297.81,A -85,B 0,C 180,E1 1813.458,E2 1813.458} C_VEL
LIN {X 0,Y 583.938,Z 297.81,A -85,B 0,C 180,E1 1818.076,E2 1818.076} C_VEL
LIN {X 0,Y 583.808,Z 297.81,A -85,B 0,C 180,E1 1822.823,E2 1822.823} C_VEL
LIN {X 0,Y 583.721,Z 297.81,A -85,B 0,C 180,E1 1828.486,E2 1828.486} C_VEL
LIN {X 0,Y 583.823,Z 297.81,A -85,B 0,C 180,E1 1834.667,E2 1834.667} C_VEL
LIN {X 0,Y 584.127,Z 298.516,A -85,B 0,C 180,E1 1837.5,E2 1837.5} C_VEL
LIN {X 0,Y 584.827,Z 324.551,A -85,B 0,C 180,E1 1838.53,E2 1838.53} C_VEL
LIN {X 0,Y 584.516,Z 348.064,A -85,B 0,C 180,E1 1840.084,E2 1840.084} C_VEL
LIN {X 0,Y 584.389,Z 366.922,A -85,B 0,C 180,E1 1842.003,E2 1842.003} C_VEL
LIN {X 0,Y 584.264,Z 381.236,A -85,B 0,C 180,E1 1844.228,E2 1844.228} C_VEL
LIN {X 0,Y 584.197,Z 389.666,A -85,B 0,C 180,E1 1846.339,E2 1846.339} C_VEL
LIN {X 0,Y 584.215,Z 394.159,A -85,B 0,C 180,E1 1848.525,E2 1848.525} C_VEL
LIN {X 0,Y 584.122,Z 394.676,A -85,B 0,C 180,E1 1850.823,E2 1850.823} C_VEL
LIN {X 0,Y 584.201,Z 389.723,A -85,B 0,C 180,E1 1853.553,E2 1853.553} C_VEL
LIN {X 0,Y 584.32,Z 379.546,A -85,B 0,C 180,E1 1856.004,E2 1856.004} C_VEL
LIN {X 0,Y 584.394,Z 364.651,A -85,B 0,C 180,E1 1858.183,E2 1858.183} C_VEL
LIN {X 0,Y 584.6,Z 344.067,A -85,B 0,C 180,E1 1860.145,E2 1860.145} C_VEL
LIN {X 0,Y 584.781,Z 320.29,A -85,B 0,C 180,E1 1861.594,E2 1861.594} C_VEL
LIN {X 0,Y 584.164,Z 297.81,A -85,B 0,C 180,E1 1862.43,E2 1862.43} C_VEL
LIN {X 0,Y 583.825,Z 297.81,A -85,B 0,C 180,E1 1868.786,E2 1868.786} C_VEL
LIN {X 0,Y 583.96,Z 297.81,A -85,B 0,C 180,E1 1873.487,E2 1873.487} C_VEL
LIN {X 0,Y 583.935,Z 297.81,A -85,B 0,C 180,E1 1879.579,E2 1879.579} C_VEL
LIN {X 0,Y 584.03,Z 297.81,A -85,B 0,C 180,E1 1883.477,E2 1883.477} C_VEL
LIN {X 0,Y 584.754,Z 322.958,A -85,B 0,C 180,E1 1884.447,E2 1884.447} C_VEL
LIN {X 0,Y 584.552,Z 346.194,A -85,B 0,C 180,E1 1885.93,E2 1885.93} C_VEL
LIN {X 0,Y 584.444,Z 366.632,A -85,B 0,C 180,E1 1887.966,E2 1887.966} C_VEL
LIN {X 0,Y 584.326,Z 381.956,A -85,B 0,C 180,E1 1890.37,E2 1890.37} C_VEL
LIN {X 0,Y 584.251,Z 391.363,A -85,B 0,C 180,E1 1892.961,E2 1892.961} C_VEL
LIN {X 0,Y 584.255,Z 394.066,A -85,B 0,C 180,E1 1894.444,E2 1894.444} C_VEL
LIN {X 0,Y 584.162,Z 394.999,A -85,B 0,C 180,E1 1895.931,E2 1895.931} C_VEL
LIN {X 0,Y 584.179,Z 393.029,A -85,B 0,C 180,E1 1898.168,E2 1898.168} C_VEL
LIN {X 0,Y 584.278,Z 385.686,A -85,B 0,C 180,E1 1900.703,E2 1900.703} C_VEL
LIN {X 0,Y 584.339,Z 373.155,A -85,B 0,C 180,E1 1903.06,E2 1903.06} C_VEL
LIN {X 0,Y 584.461,Z 354.596,A -85,B 0,C 180,E1 1905.25,E2 1905.25} C_VEL
LIN {X 0,Y 584.709,Z 332.442,A -85,B 0,C 180,E1 1906.939,E2 1906.939} C_VEL
LIN {X 0,Y 584.915,Z 307.125,A -85,B 0,C 180,E1 1908.127,E2 1908.127} C_VEL
LIN {X 0,Y 584.096,Z 297.81,A -85,B 0,C 180,E1 1908.433,E2 1908.433} C_VEL
LIN {X 0,Y 583.743,Z 297.81,A -85,B 0,C 180,E1 1914.432,E2 1914.432} C_VEL
LIN {X 0,Y 583.66,Z 297.81,A -85,B 0,C 180,E1 1919.422,E2 1919.422} C_VEL
LIN {X 0,Y 583.639,Z 297.81,A -85,B 0,C 180,E1 1924.668,E2 1924.668} C_VEL
LIN {X 0,Y 583.758,Z 297.81,A -85,B 0,C 180,E1 1929.134,E2 1929.134} C_VEL
LIN {X 0,Y 583.69,Z 297.81,A -85,B 0,C 180,E1 1935.717,E2 1935.717} C_VEL
LIN {X 0,Y 583.709,Z 297.81,A -85,B 0,C 180,E1 1941.638,E2 1941.638} C_VEL
LIN {X 0,Y 583.513,Z 297.81,A -85,B 0,C 180,E1 1947.095,E2 1947.095} C_VEL
LIN {X 0,Y 583.58,Z 297.81,A -85,B 0,C 180,E1 1952.25,E2 1952.25} C_VEL
LIN {X 0,Y 583.627,Z 297.81,A -85,B 0,C 180,E1 1957.17,E2 1957.17} C_VEL
LIN {X 0,Y 583.966,Z 297.81,A -85,B 0,C 180,E1 1961.925,E2 1961.925} C_VEL
LIN {X 0,Y 583.71,Z 297.81,A -85,B 0,C 180,E1 1968.054,E2 1968.054} C_VEL
LIN {X 0,Y 584.132,Z 297.81,A -85,B 0,C 180,E1 1974.059,E2 1974.059} C_VEL
LIN {X 0,Y 583.935,Z 297.81,A -85,B 0,C 180,E1 1979.991,E2 1979.991} C_VEL
LIN {X 0,Y 583.974,Z 297.81,A -85,B 0,C 180,E1 1984.437,E2 1984.437} C_VEL
LIN {X 0,Y 583.795,Z 297.81,A -85,B 0,C 180,E1 1985.879,E2 1985.879} C_VEL
LIN {X 0,Y 579.992,Z 297.81,A -85,B 0,C 180,E1 1987.557,E2 1987.557} C_VEL
LIN {X 0,Y 575.984,Z 297.81,A -85,B 0,C 180,E1 1989.257,E2 1989.257} C_VEL
LIN {X 0,Y 575.937,Z 297.81,A -85,B 0,C 180,E1 1994.203,E2 1994.203} C_VEL
LIN {X 0,Y 575.859,Z 297.81,A -85,B 0,C 180,E1 1999.908,E2 1999.908} C_VEL
LIN {X 0,Y 575.754,Z 297.81,A -85,B 0,C 180,E1 2004.784,E2 2004.784} C_VEL
LIN {X 0,Y 575.677,Z 297.81,A -85,B 0,C 180,E1 2010.115,E2 2010.115} C_VEL
LIN {X 0,Y 575.689,Z 297.81,A -85,B 0,C 180,E1 2015.206,E2 2015.206} C_VEL
LIN {X 0,Y 575.65,Z 297.81,A -85,B 0,C 180,E1 2020.935,E2 2020.935} C_VEL
LIN {X 0,Y 575.821,Z 297.81,A -85,B 0,C 180,E1 2027.191,E2 2027.191} C_VEL
LIN {X 0,Y 575.854,Z 297.81,A -85,B 0,C 180,E1 2032.936,E2 2032.936} C_VEL
LIN {X 0,Y 575.743,Z 297.81,A -85,B 0,C 180,E1 2038.386,E2 2038.386} C_VEL
LIN {X 0,Y 575.864,Z 297.81,A -85,B 0,C 180,E1 2043.546,E2 2043.546} C_VEL
LIN {X 0,Y 576.164,Z 297.81,A -85,B 0,C 180,E1 2047.679,E2 2047.679} C_VEL
LIN {X 0,Y 578.848,Z 310.073,A -85,B 0,C 180,E1 2047.952,E2 2047.952} C_VEL
LIN {X 0,Y 578.741,Z 377.525,A -85,B 0,C 180,E1 2048.929,E2 2048.929} C_VEL
LIN {X 0,Y 578.301,Z 410.245,A -85,B 0,C 180,E1 2049.971,E2 2049.971} C_VEL
LIN {X 0,Y 577.777,Z 442.54,A -85,B 0,C 180,E1 2051.636,E2 2051.636} C_VEL
LIN {X 0,Y 577.229,Z 471.132,A -85,B 0,C 180,E1 2053.776,E2 2053.776} C_VEL
LIN {X 0,Y 576.789,Z 496.041,A -85,B 0,C 180,E1 2056.381,E2 2056.381} C_VEL
LIN {X 0,Y 576.525,Z 515.839,A -85,B 0,C 180,E1 2059.254,E2 2059.254} C_VEL
LIN {X 0,Y 576.363,Z 531.185,A -85,B 0,C 180,E1 2062.478,E2 2062.478} C_VEL
LIN {X 0,Y 576.301,Z 540.101,A -85,B 0,C 180,E1 2065.494,E2 2065.494} C_VEL
LIN {X 0,Y 576.279,Z 544.421,A -85,B 0,C 180,E1 2068.499,E2 2068.499} C_VEL
LIN {X 0,Y 576.229,Z 544.422,A -85,B 0,C 180,E1 2071.5,E2 2071.5} C_VEL
LIN {X 0,Y 576.273,Z 540.102,A -85,B 0,C 180,E1 2074.505,E2 2074.505} C_VEL
LIN {X 0,Y 576.405,Z 529.671,A -85,B 0,C 180,E1 2077.899,E2 2077.899} C_VEL
LIN {X 0,Y 576.594,Z 513.529,A -85,B 0,C 180,E1 2081.139,E2 2081.139} C_VEL
LIN {X 0,Y 576.876,Z 491.867,A -85,B 0,C 180,E1 2084.121,E2 2084.121} C_VEL
LIN {X 0,Y 577.365,Z 465.438,A -85,B 0,C 180,E1 2086.708,E2 2086.708} C_VEL
LIN {X 0,Y 577.901,Z 436.079,A -85,B 0,C 180,E1 2088.753,E2 2088.753} C_VEL
LIN {X 0,Y 578.378,Z 404.308,A -85,B 0,C 180,E1 2090.267,E2 2090.267} C_VEL
LIN {X 0,Y 578.734,Z 370.701,A -85,B 0,C 180,E1 2091.214,E2 2091.214} C_VEL
LIN {X 0,Y 578.173,Z 304.694,A -85,B 0,C 180,E1 2092.146,E2 2092.146} C_VEL
LIN {X 0,Y 576.164,Z 297.81,A -85,B 0,C 180,E1 2092.364,E2 2092.364} C_VEL
LIN {X 0,Y 575.85,Z 297.81,A -85,B 0,C 180,E1 2098.143,E2 2098.143} C_VEL
LIN {X 0,Y 575.865,Z 297.81,A -85,B 0,C 180,E1 2103.386,E2 2103.386} C_VEL
LIN {X 0,Y 575.653,Z 297.81,A -85,B 0,C 180,E1 2108.985,E2 2108.985} C_VEL
LIN {X 0,Y 575.696,Z 297.81,A -85,B 0,C 180,E1 2115.049,E2 2115.049} C_VEL
LIN {X 0,Y 575.718,Z 297.81,A -85,B 0,C 180,E1 2121.03,E2 2121.03} C_VEL
LIN {X 0,Y 575.619,Z 297.81,A -85,B 0,C 180,E1 2126.607,E2 2126.607} C_VEL
LIN {X 0,Y 575.722,Z 297.81,A -85,B 0,C 180,E1 2131.859,E2 2131.859} C_VEL
LIN {X 0,Y 575.681,Z 297.81,A -85,B 0,C 180,E1 2136.857,E2 2136.857} C_VEL
LIN {X 0,Y 575.919,Z 297.81,A -85,B 0,C 180,E1 2141.684,E2 2141.684} C_VEL
LIN {X 0,Y 575.711,Z 297.81,A -85,B 0,C 180,E1 2147.905,E2 2147.905} C_VEL
LIN {X 0,Y 576.221,Z 297.81,A -85,B 0,C 180,E1 2153.996,E2 2153.996} C_VEL
LIN {X 0,Y 575.986,Z 297.81,A -85,B 0,C 180,E1 2160.009,E2 2160.009} C_VEL
LIN {X 0,Y 575.875,Z 297.81,A -85,B 0,C 180,E1 2165.299,E2 2165.299} C_VEL
LIN {X 0,Y 575.829,Z 297.81,A -85,B 0,C 180,E1 2170.58,E2 2170.58} C_VEL
LIN {X 0,Y 575.806,Z 297.81,A -85,B 0,C 180,E1 2175.203,E2 2175.203} C_VEL
LIN {X 0,Y 575.821,Z 297.81,A -85,B 0,C 180,E1 2179.929,E2 2179.929} C_VEL
LIN {X 0,Y 575.739,Z 297.81,A -85,B 0,C 180,E1 2184.805,E2 2184.805} C_VEL
LIN {X 0,Y 575.711,Z 297.81,A -85,B 0,C 180,E1 2190.122,E2 2190.122} C_VEL
LIN {X 0,Y 575.856,Z 297.81,A -85,B 0,C 180,E1 2195.217,E2 2195.217} C_VEL
LIN {X 0,Y 576.111,Z 297.81,A -85,B 0,C 180,E1 2197.299,E2 2197.299} C_VEL
LIN {X 0,Y 577.066,Z 322.073,A -85,B 0,C 180,E1 2198.248,E2 2198.248} C_VEL
LIN {X 0,Y 576.796,Z 345.288,A -85,B 0,C 180,E1 2199.72,E2 2199.72} C_VEL
LIN {X 0,Y 576.568,Z 365.112,A -85,B 0,C 180,E1 2201.67,E2 2201.67} C_VEL
LIN {X 0,Y 576.42,Z 380.549,A -85,B 0,C 180,E1 2204.017,E2 2204.017} C_VEL
LIN {X 0,Y 576.309,Z 389.914,A -85,B 0,C 180,E1 2206.371,E2 2206.371} C_VEL
LIN {X 0,Y 576.287,Z 394.699,A -85,B 0,C 180,E1 2209.11,E2 2209.11} C_VEL
LIN {X 0,Y 576.237,Z 393.671,A -85,B 0,C 180,E1 2211.795,E2 2211.795} C_VEL
LIN {X 0,Y 576.366,Z 386.533,A -85,B 0,C 180,E1 2214.556,E2 2214.556} C_VEL
LIN {X 0,Y 576.496,Z 374.738,A -85,B 0,C 180,E1 2216.909,E2 2216.909} C_VEL
LIN {X 0,Y 576.653,Z 357.172,A -85,B 0,C 180,E1 2219.121,E2 2219.121} C_VEL
LIN {X 0,Y 576.903,Z 335.116,A -85,B 0,C 180,E1 2220.921,E2 2220.921} C_VEL
LIN {X 0,Y 577.066,Z 309.619,A -85,B 0,C 180,E1 2222.206,E2 2222.206} C_VEL
LIN {X 0,Y 576.259,Z 297.81,A -85,B 0,C 180,E1 2222.66,E2 2222.66} C_VEL
LIN {X 0,Y 575.862,Z 297.81,A -85,B 0,C 180,E1 2228.479,E2 2228.479} C_VEL
LIN {X 0,Y 576.056,Z 297.81,A -85,B 0,C 180,E1 2233.253,E2 2233.253} C_VEL
LIN {X 0,Y 576.001,Z 297.81,A -85,B 0,C 180,E1 2239.433,E2 2239.433} C_VEL
LIN {X 0,Y 576.108,Z 298.018,A -85,B 0,C 180,E1 2243.311,E2 2243.311} C_VEL
LIN {X 0,Y 577.042,Z 320.806,A -85,B 0,C 180,E1 2244.184,E2 2244.184} C_VEL
LIN {X 0,Y 576.776,Z 344.84,A -85,B 0,C 180,E1 2245.687,E2 2245.687} C_VEL
LIN {X 0,Y 576.627,Z 364.226,A -85,B 0,C 180,E1 2247.563,E2 2247.563} C_VEL
LIN {X 0,Y 576.475,Z 379.501,A -85,B 0,C 180,E1 2249.813,E2 2249.813} C_VEL
LIN {X 0,Y 576.419,Z 389.549,A -85,B 0,C 180,E1 2252.251,E2 2252.251} C_VEL
LIN {X 0,Y 576.343,Z 394.157,A -85,B 0,C 180,E1 2254.505,E2 2254.505} C_VEL
LIN {X 0,Y 576.264,Z 394.994,A -85,B 0,C 180,E1 2256.013,E2 2256.013} C_VEL
LIN {X 0,Y 576.29,Z 392.883,A -85,B 0,C 180,E1 2258.281,E2 2258.281} C_VEL
LIN {X 0,Y 576.367,Z 385.35,A -85,B 0,C 180,E1 2260.852,E2 2260.852} C_VEL
LIN {X 0,Y 576.466,Z 372.577,A -85,B 0,C 180,E1 2263.241,E2 2263.241} C_VEL
LIN {X 0,Y 576.65,Z 354.725,A -85,B 0,C 180,E1 2265.365,E2 2265.365} C_VEL
LIN {X 0,Y 576.951,Z 331.91,A -85,B 0,C 180,E1 2267.122,E2 2267.122} C_VEL
LIN {X 0,Y 577.189,Z 307.377,A -85,B 0,C 180,E1 2268.284,E2 2268.284} C_VEL
LIN {X 0,Y 576.18,Z 297.81,A -85,B 0,C 180,E1 2268.658,E2 2268.658} C_VEL
LIN {X 0,Y 575.859,Z 297.81,A -85,B 0,C 180,E1 2274.789,E2 2274.789} C_VEL
LIN {X 0,Y 575.722,Z 297.81,A -85,B 0,C 180,E1 2280.102,E2 2280.102} C_VEL
LIN {X 0,Y 575.801,Z 297.81,A -85,B 0,C 180,E1 2285.649,E2 2285.649} C_VEL
LIN {X 0,Y 575.721,Z 297.81,A -85,B 0,C 180,E1 2290.51,E2 2290.51} C_VEL
LIN {X 0,Y 575.776,Z 297.81,A -85,B 0,C 180,E1 2297.032,E2 2297.032} C_VEL
LIN {X 0,Y 575.838,Z 297.81,A -85,B 0,C 180,E1 2302.922,E2 2302.922} C_VEL
LIN {X 0,Y 575.696,Z 297.81,A -85,B 0,C 180,E1 2308.371,E2 2308.371} C_VEL
LIN {X 0,Y 575.764,Z 297.81,A -85,B 0,C 180,E1 2313.53,E2 2313.53} C_VEL
LIN {X 0,Y 576.041,Z 297.81,A -85,B 0,C 180,E1 2320.079,E2 2320.079} C_VEL
LIN {X 0,Y 575.798,Z 297.81,A -85,B 0,C 180,E1 2324.797,E2 2324.797} C_VEL
LIN {X 0,Y 575.906,Z 297.81,A -85,B 0,C 180,E1 2330.945,E2 2330.945} C_VEL
LIN {X 0,Y 575.95,Z 297.81,A -85,B 0,C 180,E1 2335.482,E2 2335.482} C_VEL
LIN {X 0,Y 576.034,Z 297.81,A -85,B 0,C 180,E1 2339.991,E2 2339.991} C_VEL
LIN {X 0,Y 575.926,Z 297.81,A -85,B 0,C 180,E1 2345.344,E2 2345.344} C_VEL
LIN {X 0,Y 575.984,Z 297.81,A -85,B 0,C 180,E1 2349.257,E2 2349.257} C_VEL
LIN {X 0,Y 571.94,Z 297.81,A -85,B 0,C 180,E1 2350.952,E2 2350.952} C_VEL
LIN {X 0,Y 568.047,Z 297.81,A -85,B 0,C 180,E1 2352.671,E2 2352.671} C_VEL
LIN {X 0,Y 568.048,Z 297.81,A -85,B 0,C 180,E1 2358.579,E2 2358.579} C_VEL
LIN {X 0,Y 567.944,Z 297.81,A -85,B 0,C 180,E1 2363.477,E2 2363.477} C_VEL
LIN {X 0,Y 567.846,Z 297.81,A -85,B 0,C 180,E1 2368.723,E2 2368.723} C_VEL
LIN {X 0,Y 567.789,Z 297.81,A -85,B 0,C 180,E1 2374.524,E2 2374.524} C_VEL
LIN {X 0,Y 567.762,Z 297.81,A -85,B 0,C 180,E1 2379.622,E2 2379.622} C_VEL
LIN {X 0,Y 567.808,Z 297.81,A -85,B 0,C 180,E1 2385.841,E2 2385.841} C_VEL
LIN {X 0,Y 567.848,Z 297.81,A -85,B 0,C 180,E1 2390.399,E2 2390.399} C_VEL
LIN {X 0,Y 567.745,Z 297.81,A -85,B 0,C 180,E1 2395.467,E2 2395.467} C_VEL
LIN {X 0,Y 567.815,Z 297.81,A -85,B 0,C 180,E1 2401.265,E2 2401.265} C_VEL
LIN {X 0,Y 568.244,Z 297.81,A -85,B 0,C 180,E1 2407.341,E2 2407.341} C_VEL
LIN {X 0,Y 571.544,Z 310.243,A -85,B 0,C 180,E1 2407.657,E2 2407.657} C_VEL
LIN {X 0,Y 571.375,Z 377.981,A -85,B 0,C 180,E1 2408.656,E2 2408.656} C_VEL
LIN {X 0,Y 570.82,Z 411.456,A -85,B 0,C 180,E1 2409.748,E2 2409.748} C_VEL
LIN {X 0,Y 570.192,Z 442.536,A -85,B 0,C 180,E1 2411.383,E2 2411.383} C_VEL
LIN {X 0,Y 569.592,Z 471.132,A -85,B 0,C 180,E1 2413.552,E2 2413.552} C_VEL
LIN {X 0,Y 569.014,Z 496.04,A -85,B 0,C 180,E1 2416.191,E2 2416.191} C_VEL
LIN {X 0,Y 568.68,Z 515.316,A -85,B 0,C 180,E1 2419.011,E2 2419.011} C_VEL
LIN {X 0,Y 568.481,Z 531.184,A -85,B 0,C 180,E1 2422.373,E2 2422.373} C_VEL
LIN {X 0,Y 568.41,Z 540.1,A -85,B 0,C 180,E1 2425.432,E2 2425.432} C_VEL
LIN {X 0,Y 568.393,Z 544.421,A -85,B 0,C 180,E1 2428.478,E2 2428.478} C_VEL
LIN {X 0,Y 568.348,Z 544.421,A -85,B 0,C 180,E1 2431.521,E2 2431.521} C_VEL
LIN {X 0,Y 568.425,Z 538.84,A -85,B 0,C 180,E1 2435.116,E2 2435.116} C_VEL
LIN {X 0,Y 568.532,Z 528.141,A -85,B 0,C 180,E1 2438.394,E2 2438.394} C_VEL
LIN {X 0,Y 568.785,Z 512.034,A -85,B 0,C 180,E1 2441.536,E2 2441.536} C_VEL
LIN {X 0,Y 569.153,Z 490.67,A -85,B 0,C 180,E1 2444.456,E2 2444.456} C_VEL
LIN {X 0,Y 569.733,Z 463.974,A -85,B 0,C 180,E1 2447.064,E2 2447.064} C_VEL
LIN {X 0,Y 570.382,Z 434.375,A -85,B 0,C 180,E1 2449.11,E2 2449.11} C_VEL
LIN {X 0,Y 571.02,Z 402.045,A -85,B 0,C 180,E1 2450.622,E2 2450.622} C_VEL
LIN {X 0,Y 571.392,Z 368.477,A -85,B 0,C 180,E1 2451.546,E2 2451.546} C_VEL
LIN {X 0,Y 570.882,Z 306.565,A -85,B 0,C 180,E1 2452.419,E2 2452.419} C_VEL
LIN {X 0,Y 568.224,Z 297.81,A -85,B 0,C 180,E1 2452.665,E2 2452.665} C_VEL
LIN {X 0,Y 567.84,Z 297.81,A -85,B 0,C 180,E1 2458.739,E2 2458.739} C_VEL
LIN {X 0,Y 567.78,Z 297.81,A -85,B 0,C 180,E1 2464.538,E2 2464.538} C_VEL
LIN {X 0,Y 567.706,Z 297.81,A -85,B 0,C 180,E1 2469.637,E2 2469.637} C_VEL
LIN {X 0,Y 567.734,Z 297.81,A -85,B 0,C 180,E1 2475.859,E2 2475.859} C_VEL
LIN {X 0,Y 567.81,Z 297.81,A -85,B 0,C 180,E1 2480.416,E2 2480.416} C_VEL
LIN {X 0,Y 567.68,Z 297.81,A -85,B 0,C 180,E1 2485.49,E2 2485.49} C_VEL
LIN {X 0,Y 567.77,Z 297.81,A -85,B 0,C 180,E1 2491.289,E2 2491.289} C_VEL
LIN {X 0,Y 567.803,Z 297.81,A -85,B 0,C 180,E1 2496.516,E2 2496.516} C_VEL
LIN {X 0,Y 568.031,Z 297.81,A -85,B 0,C 180,E1 2501.42,E2 2501.42} C_VEL
LIN {X 0,Y 567.668,Z 297.81,A -85,B 0,C 180,E1 2506.168,E2 2506.168} C_VEL
LIN {X 0,Y 567.939,Z 297.81,A -85,B 0,C 180,E1 2510.836,E2 2510.836} C_VEL
LIN {X 0,Y 568.058,Z 297.81,A -85,B 0,C 180,E1 2515.438,E2 2515.438} C_VEL
LIN {X 0,Y 568.111,Z 297.81,A -85,B 0,C 180,E1 2520.009,E2 2520.009} C_VEL
LIN {X 0,Y 568.073,Z 297.81,A -85,B 0,C 180,E1 2524.58,E2 2524.58} C_VEL
LIN {X 0,Y 568.104,Z 297.81,A -85,B 0,C 180,E1 2529.18,E2 2529.18} C_VEL
LIN {X 0,Y 568.091,Z 297.81,A -85,B 0,C 180,E1 2533.841,E2 2533.841} C_VEL
LIN {X 0,Y 568.056,Z 297.81,A -85,B 0,C 180,E1 2538.599,E2 2538.599} C_VEL
LIN {X 0,Y 567.906,Z 297.81,A -85,B 0,C 180,E1 2543.5,E2 2543.5} C_VEL
LIN {X 0,Y 567.862,Z 297.81,A -85,B 0,C 180,E1 2548.728,E2 2548.728} C_VEL
LIN {X 0,Y 567.929,Z 297.81,A -85,B 0,C 180,E1 2554.546,E2 2554.546} C_VEL
LIN {X 0,Y 568.171,Z 297.875,A -85,B 0,C 180,E1 2557.126,E2 2557.126} C_VEL
LIN {X 0,Y 569.364,Z 316.28,A -85,B 0,C 180,E1 2557.812,E2 2557.812} C_VEL
LIN {X 0,Y 569.062,Z 341.022,A -85,B 0,C 180,E1 2559.25,E2 2559.25} C_VEL
LIN {X 0,Y 568.755,Z 361.968,A -85,B 0,C 180,E1 2561.179,E2 2561.179} C_VEL
LIN {X 0,Y 568.616,Z 377.829,A -85,B 0,C 180,E1 2563.426,E2 2563.426} C_VEL
LIN {X 0,Y 568.464,Z 388.323,A -85,B 0,C 180,E1 2565.8,E2 2565.8} C_VEL
LIN {X 0,Y 568.355,Z 394.078,A -85,B 0,C 180,E1 2568.414,E2 2568.414} C_VEL
LIN {X 0,Y 568.312,Z 394.447,A -85,B 0,C 180,E1 2571.163,E2 2571.163} C_VEL
LIN {X 0,Y 568.419,Z 389.579,A -85,B 0,C 180,E1 2573.702,E2 2573.702} C_VEL
LIN {X 0,Y 568.561,Z 379.775,A -85,B 0,C 180,E1 2576.128,E2 2576.128} C_VEL
LIN {X 0,Y 568.717,Z 364.542,A -85,B 0,C 180,E1 2578.424,E2 2578.424} C_VEL
LIN {X 0,Y 568.988,Z 344.979,A -85,B 0,C 180,E1 2580.357,E2 2580.357} C_VEL
LIN {X 0,Y 569.278,Z 320.362,A -85,B 0,C 180,E1 2581.911,E2 2581.911} C_VEL
LIN {X 0,Y 568.367,Z 297.81,A -85,B 0,C 180,E1 2582.857,E2 2582.857} C_VEL
LIN {X 0,Y 568.029,Z 297.81,A -85,B 0,C 180,E1 2589.797,E2 2589.797} C_VEL
LIN {X 0,Y 567.916,Z 297.81,A -85,B 0,C 180,E1 2594.591,E2 2594.591} C_VEL
LIN {X 0,Y 568.01,Z 297.81,A -85,B 0,C 180,E1 2600.828,E2 2600.828} C_VEL
LIN {X 0,Y 568.19,Z 297.81,A -85,B 0,C 180,E1 2603.116,E2 2603.116} C_VEL
LIN {X 0,Y 569.307,Z 318.559,A -85,B 0,C 180,E1 2603.914,E2 2603.914} C_VEL
LIN {X 0,Y 569.009,Z 342.281,A -85,B 0,C 180,E1 2605.343,E2 2605.343} C_VEL
LIN {X 0,Y 568.797,Z 363.337,A -85,B 0,C 180,E1 2607.339,E2 2607.339} C_VEL
LIN {X 0,Y 568.636,Z 378.91,A -85,B 0,C 180,E1 2609.62,E2 2609.62} C_VEL
LIN {X 0,Y 568.54,Z 389.792,A -85,B 0,C 180,E1 2612.282,E2 2612.282} C_VEL
LIN {X 0,Y 568.447,Z 394.249,A -85,B 0,C 180,E1 2614.568,E2 2614.568} C_VEL
LIN {X 0,Y 568.357,Z 394.976,A -85,B 0,C 180,E1 2616.097,E2 2616.097} C_VEL
LIN {X 0,Y 568.419,Z 392.717,A -85,B 0,C 180,E1 2618.396,E2 2618.396} C_VEL
LIN {X 0,Y 568.469,Z 384.805,A -85,B 0,C 180,E1 2621.057,E2 2621.057} C_VEL
LIN {X 0,Y 568.613,Z 372.001,A -85,B 0,C 180,E1 2623.428,E2 2623.428} C_VEL
LIN {X 0,Y 568.806,Z 353.813,A -85,B 0,C 180,E1 2625.582,E2 2625.582} C_VEL
LIN {X 0,Y 569.187,Z 331.586,A -85,B 0,C 180,E1 2627.295,E2 2627.295} C_VEL
LIN {X 0,Y 569.457,Z 306.112,A -85,B 0,C 180,E1 2628.499,E2 2628.499} C_VEL
LIN {X 0,Y 568.284,Z 297.81,A -85,B 0,C 180,E1 2628.838,E2 2628.838} C_VEL
LIN {X 0,Y 567.866,Z 297.81,A -85,B 0,C 180,E1 2635.354,E2 2635.354} C_VEL
LIN {X 0,Y 567.787,Z 297.81,A -85,B 0,C 180,E1 2641.718,E2 2641.718} C_VEL
LIN {X 0,Y 568.031,Z 297.81,A -85,B 0,C 180,E1 2647.663,E2 2647.663} C_VEL
LIN {X 0,Y 567.703,Z 297.81,A -85,B 0,C 180,E1 2654.121,E2 2654.121} C_VEL
LIN {X 0,Y 567.827,Z 297.81,A -85,B 0,C 180,E1 2660.358,E2 2660.358} C_VEL
LIN {X 0,Y 567.695,Z 297.81,A -85,B 0,C 180,E1 2665.489,E2 2665.489} C_VEL
LIN {X 0,Y 567.809,Z 297.81,A -85,B 0,C 180,E1 2669.661,E2 2669.661} C_VEL
LIN {X 0,Y 567.889,Z 297.81,A -85,B 0,C 180,E1 2674.828,E2 2674.828} C_VEL
LIN {X 0,Y 568.075,Z 297.81,A -85,B 0,C 180,E1 2679.788,E2 2679.788} C_VEL
LIN {X 0,Y 567.906,Z 297.81,A -85,B 0,C 180,E1 2684.58,E2 2684.58} C_VEL
LIN {X 0,Y 568,Z 297.81,A -85,B 0,C 180,E1 2690.818,E2 2690.818} C_VEL
LIN {X 0,Y 568.06,Z 297.81,A -85,B 0,C 180,E1 2695.419,E2 2695.419} C_VEL
LIN {X 0,Y 568.158,Z 297.81,A -85,B 0,C 180,E1 2699.991,E2 2699.991} C_VEL
LIN {X 0,Y 568.143,Z 297.81,A -85,B 0,C 180,E1 2704.561,E2 2704.561} C_VEL
LIN {X 0,Y 568.087,Z 297.81,A -85,B 0,C 180,E1 2709.24,E2 2709.24} C_VEL
LIN {X 0,Y 568.047,Z 297.81,A -85,B 0,C 180,E1 2712.671,E2 2712.671} C_VEL
LIN {X 0,Y 565.466,Z 297.81,A -85,B 0,C 180,E1 2713.968,E2 2713.968} C_VEL
LIN {X 0,Y 560.066,Z 297.81,A -85,B 0,C 180,E1 2715.911,E2 2715.911} C_VEL
LIN {X 0,Y 559.974,Z 297.81,A -85,B 0,C 180,E1 2716.135,E2 2716.135} C_VEL
LIN {X 0,Y 560.035,Z 297.81,A -85,B 0,C 180,E1 2720.495,E2 2720.495} C_VEL
LIN {X 0,Y 559.894,Z 297.81,A -85,B 0,C 180,E1 2725.535,E2 2725.535} C_VEL
LIN {X 0,Y 559.874,Z 297.81,A -85,B 0,C 180,E1 2730.793,E2 2730.793} C_VEL
LIN {X 0,Y 559.801,Z 297.81,A -85,B 0,C 180,E1 2736.362,E2 2736.362} C_VEL
LIN {X 0,Y 559.78,Z 297.81,A -85,B 0,C 180,E1 2742.359,E2 2742.359} C_VEL
LIN {X 0,Y 559.904,Z 297.81,A -85,B 0,C 180,E1 2747.64,E2 2747.64} C_VEL
LIN {X 0,Y 559.976,Z 297.81,A -85,B 0,C 180,E1 2753.929,E2 2753.929} C_VEL
LIN {X 0,Y 559.976,Z 297.81,A -85,B 0,C 180,E1 2759.562,E2 2759.562} C_VEL
LIN {X 0,Y 560.227,Z 297.81,A -85,B 0,C 180,E1 2766.169,E2 2766.169} C_VEL
LIN {X 0,Y 560.316,Z 297.81,A -85,B 0,C 180,E1 2767.041,E2 2767.041} C_VEL
LIN {X 0,Y 564.181,Z 312.881,A -85,B 0,C 180,E1 2767.403,E2 2767.403} C_VEL
LIN {X 0,Y 564.032,Z 377.98,A -85,B 0,C 180,E1 2768.364,E2 2768.364} C_VEL
LIN {X 0,Y 563.391,Z 411.459,A -85,B 0,C 180,E1 2769.469,E2 2769.469} C_VEL
LIN {X 0,Y 562.653,Z 442.544,A -85,B 0,C 180,E1 2771.125,E2 2771.125} C_VEL
LIN {X 0,Y 561.896,Z 471.133,A -85,B 0,C 180,E1 2773.32,E2 2773.32} C_VEL
LIN {X 0,Y 561.248,Z 496.039,A -85,B 0,C 180,E1 2775.996,E2 2775.996} C_VEL
LIN {X 0,Y 560.866,Z 515.317,A -85,B 0,C 180,E1 2778.856,E2 2778.856} C_VEL
LIN {X 0,Y 560.626,Z 531.184,A -85,B 0,C 180,E1 2782.265,E2 2782.265} C_VEL
LIN {X 0,Y 560.511,Z 540.099,A -85,B 0,C 180,E1 2785.367,E2 2785.367} C_VEL
LIN {X 0,Y 560.489,Z 544.42,A -85,B 0,C 180,E1 2788.457,E2 2788.457} C_VEL
LIN {X 0,Y 560.445,Z 544.421,A -85,B 0,C 180,E1 2791.542,E2 2791.542} C_VEL
LIN {X 0,Y 560.526,Z 538.904,A -85,B 0,C 180,E1 2795.162,E2 2795.162} C_VEL
LIN {X 0,Y 560.647,Z 528.141,A -85,B 0,C 180,E1 2798.513,E2 2798.513} C_VEL
LIN {X 0,Y 560.903,Z 511.202,A -85,B 0,C 180,E1 2801.837,E2 2801.837} C_VEL
LIN {X 0,Y 561.393,Z 489.822,A -85,B 0,C 180,E1 2804.756,E2 2804.756} C_VEL
LIN {X 0,Y 562.096,Z 463.973,A -85,B 0,C 180,E1 2807.303,E2 2807.303} C_VEL
LIN {X 0,Y 562.861,Z 434.441,A -85,B 0,C 180,E1 2809.371,E2 2809.371} C_VEL
LIN {X 0,Y 563.602,Z 402.732,A -85,B 0,C 180,E1 2810.881,E2 2810.881} C_VEL
LIN {X 0,Y 564.066,Z 368.458,A -85,B 0,C 180,E1 2811.84,E2 2811.84} C_VEL
LIN {X 0,Y 563.44,Z 308.25,A -85,B 0,C 180,E1 2812.681,E2 2812.681} C_VEL
LIN {X 0,Y 560.264,Z 297.81,A -85,B 0,C 180,E1 2812.957,E2 2812.957} C_VEL
LIN {X 0,Y 559.901,Z 297.81,A -85,B 0,C 180,E1 2819.02,E2 2819.02} C_VEL
LIN {X 0,Y 559.897,Z 297.81,A -85,B 0,C 180,E1 2824.47,E2 2824.47} C_VEL
LIN {X 0,Y 559.706,Z 297.81,A -85,B 0,C 180,E1 2830.319,E2 2830.319} C_VEL
LIN {X 0,Y 559.782,Z 297.81,A -85,B 0,C 180,E1 2835.514,E2 2835.514} C_VEL
LIN {X 0,Y 559.86,Z 297.81,A -85,B 0,C 180,E1 2841.41,E2 2841.41} C_VEL
LIN {X 0,Y 559.756,Z 297.81,A -85,B 0,C 180,E1 2846.688,E2 2846.688} C_VEL
LIN {X 0,Y 559.851,Z 297.81,A -85,B 0,C 180,E1 2850.987,E2 2850.987} C_VEL
LIN {X 0,Y 559.917,Z 297.81,A -85,B 0,C 180,E1 2856.392,E2 2856.392} C_VEL
LIN {X 0,Y 560.09,Z 297.81,A -85,B 0,C 180,E1 2861.147,E2 2861.147} C_VEL
LIN {X 0,Y 559.771,Z 297.81,A -85,B 0,C 180,E1 2866.038,E2 2866.038} C_VEL
LIN {X 0,Y 560.034,Z 297.81,A -85,B 0,C 180,E1 2870.706,E2 2870.706} C_VEL
LIN {X 0,Y 560.171,Z 297.81,A -85,B 0,C 180,E1 2875.374,E2 2875.374} C_VEL
LIN {X 0,Y 560.21,Z 297.81,A -85,B 0,C 180,E1 2880.01,E2 2880.01} C_VEL
LIN {X 0,Y 560.164,Z 297.81,A -85,B 0,C 180,E1 2884.645,E2 2884.645} C_VEL
LIN {X 0,Y 560.185,Z 297.81,A -85,B 0,C 180,E1 2889.311,E2 2889.311} C_VEL
LIN {X 0,Y 560.139,Z 297.81,A -85,B 0,C 180,E1 2894.112,E2 2894.112} C_VEL
LIN {X 0,Y 560.034,Z 297.81,A -85,B 0,C 180,E1 2899.429,E2 2899.429} C_VEL
LIN {X 0,Y 559.969,Z 297.81,A -85,B 0,C 180,E1 2903.853,E2 2903.853} C_VEL
LIN {X 0,Y 559.927,Z 297.81,A -85,B 0,C 180,E1 2909.031,E2 2909.031} C_VEL
LIN {X 0,Y 560.043,Z 297.81,A -85,B 0,C 180,E1 2914.473,E2 2914.473} C_VEL
LIN {X 0,Y 560.263,Z 298.191,A -85,B 0,C 180,E1 2916.912,E2 2916.912} C_VEL
LIN {X 0,Y 561.687,Z 314.389,A -85,B 0,C 180,E1 2917.541,E2 2917.541} C_VEL
LIN {X 0,Y 561.328,Z 339.456,A -85,B 0,C 180,E1 2918.986,E2 2918.986} C_VEL
LIN {X 0,Y 560.95,Z 360.552,A -85,B 0,C 180,E1 2920.898,E2 2920.898} C_VEL
LIN {X 0,Y 560.716,Z 376.377,A -85,B 0,C 180,E1 2923.074,E2 2923.074} C_VEL
LIN {X 0,Y 560.599,Z 387.786,A -85,B 0,C 180,E1 2925.585,E2 2925.585} C_VEL
LIN {X 0,Y 560.477,Z 393.098,A -85,B 0,C 180,E1 2927.695,E2 2927.695} C_VEL
LIN {X 0,Y 560.361,Z 394.96,A -85,B 0,C 180,E1 2929.738,E2 2929.738} C_VEL
LIN {X 0,Y 560.461,Z 393.055,A -85,B 0,C 180,E1 2932.243,E2 2932.243} C_VEL
LIN {X 0,Y 560.595,Z 385.99,A -85,B 0,C 180,E1 2934.826,E2 2934.826} C_VEL
LIN {X 0,Y 560.806,Z 372.61,A -85,B 0,C 180,E1 2937.443,E2 2937.443} C_VEL
LIN {X 0,Y 561.084,Z 353.775,A -85,B 0,C 180,E1 2939.722,E2 2939.722} C_VEL
LIN {X 0,Y 561.45,Z 330.755,A -85,B 0,C 180,E1 2941.507,E2 2941.507} C_VEL
LIN {X 0,Y 561.519,Z 305.702,A -85,B 0,C 180,E1 2942.71,E2 2942.71} C_VEL
LIN {X 0,Y 560.421,Z 297.81,A -85,B 0,C 180,E1 2943.084,E2 2943.084} C_VEL
LIN {X 0,Y 560.092,Z 297.81,A -85,B 0,C 180,E1 2949.498,E2 2949.498} C_VEL
LIN {X 0,Y 560.022,Z 297.81,A -85,B 0,C 180,E1 2954.369,E2 2954.369} C_VEL
LIN {X 0,Y 560.106,Z 297.81,A -85,B 0,C 180,E1 2960.698,E2 2960.698} C_VEL
LIN {X 0,Y 560.264,Z 297.923,A -85,B 0,C 180,E1 2962.933,E2 2962.933} C_VEL
LIN {X 0,Y 561.604,Z 316.863,A -85,B 0,C 180,E1 2963.66,E2 2963.66} C_VEL
LIN {X 0,Y 561.243,Z 341.61,A -85,B 0,C 180,E1 2965.144,E2 2965.144} C_VEL
LIN {X 0,Y 560.966,Z 362.403,A -85,B 0,C 180,E1 2967.109,E2 2967.109} C_VEL
LIN {X 0,Y 560.762,Z 378.315,A -85,B 0,C 180,E1 2969.422,E2 2969.422} C_VEL
LIN {X 0,Y 560.641,Z 388.913,A -85,B 0,C 180,E1 2971.928,E2 2971.928} C_VEL
LIN {X 0,Y 560.535,Z 394.34,A -85,B 0,C 180,E1 2974.633,E2 2974.633} C_VEL
LIN {X 0,Y 560.469,Z 394.958,A -85,B 0,C 180,E1 2976.183,E2 2976.183} C_VEL
LIN {X 0,Y 560.533,Z 392.549,A -85,B 0,C 180,E1 2978.515,E2 2978.515} C_VEL
LIN {X 0,Y 560.579,Z 384.278,A -85,B 0,C 180,E1 2981.254,E2 2981.254} C_VEL
LIN {X 0,Y 560.727,Z 371.422,A -85,B 0,C 180,E1 2983.62,E2 2983.62} C_VEL
LIN {X 0,Y 561.018,Z 352.906,A -85,B 0,C 180,E1 2985.804,E2 2985.804} C_VEL
LIN {X 0,Y 561.46,Z 330.52,A -85,B 0,C 180,E1 2987.518,E2 2987.518} C_VEL
LIN {X 0,Y 561.603,Z 305.416,A -85,B 0,C 180,E1 2988.709,E2 2988.709} C_VEL
LIN {X 0,Y 560.381,Z 297.81,A -85,B 0,C 180,E1 2989.006,E2 2989.006} C_VEL
LIN {X 0,Y 559.937,Z 297.81,A -85,B 0,C 180,E1 2995.544,E2 2995.544} C_VEL
LIN {X 0,Y 559.87,Z 297.81,A -85,B 0,C 180,E1 3000.804,E2 3000.804} C_VEL
LIN {X 0,Y 560.037,Z 297.81,A -85,B 0,C 180,E1 3006.355,E2 3006.355} C_VEL
LIN {X 0,Y 559.74,Z 297.81,A -85,B 0,C 180,E1 3012.375,E2 3012.375} C_VEL
LIN {X 0,Y 559.867,Z 297.81,A -85,B 0,C 180,E1 3017.623,E2 3017.623} C_VEL
LIN {X 0,Y 559.95,Z 297.81,A -85,B 0,C 180,E1 3023.947,E2 3023.947} C_VEL
LIN {X 0,Y 559.927,Z 297.81,A -85,B 0,C 180,E1 3029.587,E2 3029.587} C_VEL
LIN {X 0,Y 559.94,Z 297.81,A -85,B 0,C 180,E1 3034.445,E2 3034.445} C_VEL
LIN {X 0,Y 560.155,Z 297.81,A -85,B 0,C 180,E1 3040.539,E2 3040.539} C_VEL
LIN {X 0,Y 559.859,Z 297.81,A -85,B 0,C 180,E1 3045.951,E2 3045.951} C_VEL
LIN {X 0,Y 560.094,Z 297.81,A -85,B 0,C 180,E1 3050.687,E2 3050.687} C_VEL
LIN {X 0,Y 560.172,Z 297.81,A -85,B 0,C 180,E1 3055.355,E2 3055.355} C_VEL
LIN {X 0,Y 560.257,Z 297.81,A -85,B 0,C 180,E1 3059.99,E2 3059.99} C_VEL
LIN {X 0,Y 560.219,Z 297.81,A -85,B 0,C 180,E1 3064.704,E2 3064.704} C_VEL
LIN {X 0,Y 560.207,Z 297.81,A -85,B 0,C 180,E1 3069.291,E2 3069.291} C_VEL
LIN {X 0,Y 560.166,Z 297.81,A -85,B 0,C 180,E1 3074.12,E2 3074.12} C_VEL
LIN {X 0,Y 559.974,Z 297.81,A -85,B 0,C 180,E1 3076.135,E2 3076.135} C_VEL
LIN {X 0,Y 558.753,Z 297.81,A -85,B 0,C 180,E1 3077.018,E2 3077.018} C_VEL
LIN {X 0,Y 552.211,Z 297.81,A -85,B 0,C 180,E1 3079.423,E2 3079.423} C_VEL
LIN {X 0,Y 552.1,Z 297.81,A -85,B 0,C 180,E1 3079.651,E2 3079.651} C_VEL
LIN {X 0,Y 552.011,Z 297.81,A -85,B 0,C 180,E1 3085.564,E2 3085.564} C_VEL
LIN {X 0,Y 551.929,Z 297.81,A -85,B 0,C 180,E1 3091.286,E2 3091.286} C_VEL
LIN {X 0,Y 551.818,Z 297.81,A -85,B 0,C 180,E1 3096.974,E2 3096.974} C_VEL
LIN {X 0,Y 551.888,Z 297.81,A -85,B 0,C 180,E1 3103.111,E2 3103.111} C_VEL
LIN {X 0,Y 552,Z 297.81,A -85,B 0,C 180,E1 3108.997,E2 3108.997} C_VEL
LIN {X 0,Y 551.951,Z 297.81,A -85,B 0,C 180,E1 3115.088,E2 3115.088} C_VEL
LIN {X 0,Y 552.014,Z 297.81,A -85,B 0,C 180,E1 3121,E2 3121} C_VEL
LIN {X 0,Y 552.397,Z 297.81,A -85,B 0,C 180,E1 3126.799,E2 3126.799} C_VEL
LIN {X 0,Y 556.673,Z 312.684,A -85,B 0,C 180,E1 3127.148,E2 3127.148} C_VEL
LIN {X 0,Y 556.514,Z 377.703,A -85,B 0,C 180,E1 3128.109,E2 3128.109} C_VEL
LIN {X 0,Y 555.865,Z 411.94,A -85,B 0,C 180,E1 3129.23,E2 3129.23} C_VEL
LIN {X 0,Y 555.125,Z 442.73,A -85,B 0,C 180,E1 3130.872,E2 3130.872} C_VEL
LIN {X 0,Y 554.263,Z 471.133,A -85,B 0,C 180,E1 3133.084,E2 3133.084} C_VEL
LIN {X 0,Y 553.484,Z 496.038,A -85,B 0,C 180,E1 3135.796,E2 3135.796} C_VEL
LIN {X 0,Y 553.021,Z 515.827,A -85,B 0,C 180,E1 3138.789,E2 3138.789} C_VEL
LIN {X 0,Y 552.734,Z 531.183,A -85,B 0,C 180,E1 3142.154,E2 3142.154} C_VEL
LIN {X 0,Y 552.628,Z 540.099,A -85,B 0,C 180,E1 3145.301,E2 3145.301} C_VEL
LIN {X 0,Y 552.585,Z 544.42,A -85,B 0,C 180,E1 3148.435,E2 3148.435} C_VEL
LIN {X 0,Y 552.542,Z 544.42,A -85,B 0,C 180,E1 3151.564,E2 3151.564} C_VEL
LIN {X 0,Y 552.634,Z 538.905,A -85,B 0,C 180,E1 3155.236,E2 3155.236} C_VEL
LIN {X 0,Y 552.785,Z 528.142,A -85,B 0,C 180,E1 3158.635,E2 3158.635} C_VEL
LIN {X 0,Y 553.072,Z 512.399,A -85,B 0,C 180,E1 3161.807,E2 3161.807} C_VEL
LIN {X 0,Y 553.614,Z 490.794,A -85,B 0,C 180,E1 3164.856,E2 3164.856} C_VEL
LIN {X 0,Y 554.415,Z 465.43,A -85,B 0,C 180,E1 3167.421,E2 3167.421} C_VEL
LIN {X 0,Y 555.297,Z 435.731,A -85,B 0,C 180,E1 3169.566,E2 3169.566} C_VEL
LIN {X 0,Y 556.033,Z 404.38,A -85,B 0,C 180,E1 3171.074,E2 3171.074} C_VEL
LIN {X 0,Y 556.513,Z 370.164,A -85,B 0,C 180,E1 3172.047,E2 3172.047} C_VEL
LIN {X 0,Y 555.88,Z 309.771,A -85,B 0,C 180,E1 3172.907,E2 3172.907} C_VEL
LIN {X 0,Y 552.309,Z 297.81,A -85,B 0,C 180,E1 3173.225,E2 3173.225} C_VEL
LIN {X 0,Y 551.985,Z 297.81,A -85,B 0,C 180,E1 3179.477,E2 3179.477} C_VEL
LIN {X 0,Y 551.924,Z 297.81,A -85,B 0,C 180,E1 3185.04,E2 3185.04} C_VEL
LIN {X 0,Y 551.831,Z 297.81,A -85,B 0,C 180,E1 3191.017,E2 3191.017} C_VEL
LIN {X 0,Y 551.919,Z 297.81,A -85,B 0,C 180,E1 3196.892,E2 3196.892} C_VEL
LIN {X 0,Y 551.932,Z 297.81,A -85,B 0,C 180,E1 3203.034,E2 3203.034} C_VEL
LIN {X 0,Y 551.89,Z 297.81,A -85,B 0,C 180,E1 3208.711,E2 3208.711} C_VEL
LIN {X 0,Y 552.081,Z 297.81,A -85,B 0,C 180,E1 3214.419,E2 3214.419} C_VEL
LIN {X 0,Y 552.177,Z 297.81,A -85,B 0,C 180,E1 3220.866,E2 3220.866} C_VEL
LIN {X 0,Y 551.877,Z 297.81,A -85,B 0,C 180,E1 3225.764,E2 3225.764} C_VEL
LIN {X 0,Y 552.121,Z 297.81,A -85,B 0,C 180,E1 3230.571,E2 3230.571} C_VEL
LIN {X 0,Y 552.306,Z 297.81,A -85,B 0,C 180,E1 3235.308,E2 3235.308} C_VEL
LIN {X 0,Y 552.313,Z 297.81,A -85,B 0,C 180,E1 3240.01,E2 3240.01} C_VEL
LIN {X 0,Y 552.252,Z 297.81,A -85,B 0,C 180,E1 3244.712,E2 3244.712} C_VEL
LIN {X 0,Y 552.15,Z 297.81,A -85,B 0,C 180,E1 3250.311,E2 3250.311} C_VEL
LIN {X 0,Y 552.091,Z 297.81,A -85,B 0,C 180,E1 3255.873,E2 3255.873} C_VEL
LIN {X 0,Y 552.045,Z 297.81,A -85,B 0,C 180,E1 3261.663,E2 3261.663} C_VEL
LIN {X 0,Y 551.99,Z 297.81,A -85,B 0,C 180,E1 3267.705,E2 3267.705} C_VEL
LIN {X 0,Y 552.124,Z 297.81,A -85,B 0,C 180,E1 3273.148,E2 3273.148} C_VEL
LIN {X 0,Y 552.283,Z 297.81,A -85,B 0,C 180,E1 3276.611,E2 3276.611} C_VEL
LIN {X 0,Y 554.104,Z 313.535,A -85,B 0,C 180,E1 3277.253,E2 3277.253} C_VEL
LIN {X 0,Y 553.749,Z 336.919,A -85,B 0,C 180,E1 3278.552,E2 3278.552} C_VEL
LIN {X 0,Y 553.298,Z 357.295,A -85,B 0,C 180,E1 3280.324,E2 3280.324} C_VEL
LIN {X 0,Y 552.891,Z 374.094,A -85,B 0,C 180,E1 3282.532,E2 3282.532} C_VEL
LIN {X 0,Y 552.729,Z 386.836,A -85,B 0,C 180,E1 3285.236,E2 3285.236} C_VEL
LIN {X 0,Y 552.603,Z 392.866,A -85,B 0,C 180,E1 3287.518,E2 3287.518} C_VEL
LIN {X 0,Y 552.448,Z 394.996,A -85,B 0,C 180,E1 3289.908,E2 3289.908} C_VEL
LIN {X 0,Y 552.576,Z 392.878,A -85,B 0,C 180,E1 3292.386,E2 3292.386} C_VEL
LIN {X 0,Y 552.768,Z 384.58,A -85,B 0,C 180,E1 3295.272,E2 3295.272} C_VEL
LIN {X 0,Y 552.992,Z 371.366,A -85,B 0,C 180,E1 3297.792,E2 3297.792} C_VEL
LIN {X 0,Y 553.361,Z 352.967,A -85,B 0,C 180,E1 3300.013,E2 3300.013} C_VEL
LIN {X 0,Y 553.834,Z 331.391,A -85,B 0,C 180,E1 3301.709,E2 3301.709} C_VEL
LIN {X 0,Y 553.848,Z 305.356,A -85,B 0,C 180,E1 3302.964,E2 3302.964} C_VEL
LIN {X 0,Y 552.48,Z 297.81,A -85,B 0,C 180,E1 3303.328,E2 3303.328} C_VEL
LIN {X 0,Y 552.133,Z 297.81,A -85,B 0,C 180,E1 3309.189,E2 3309.189} C_VEL
LIN {X 0,Y 552.122,Z 297.81,A -85,B 0,C 180,E1 3314.139,E2 3314.139} C_VEL
LIN {X 0,Y 552.191,Z 297.81,A -85,B 0,C 180,E1 3320.563,E2 3320.563} C_VEL
LIN {X 0,Y 552.337,Z 297.81,A -85,B 0,C 180,E1 3322.692,E2 3322.692} C_VEL
LIN {X 0,Y 553.969,Z 317.053,A -85,B 0,C 180,E1 3323.451,E2 3323.451} C_VEL
LIN {X 0,Y 553.587,Z 340.538,A -85,B 0,C 180,E1 3324.843,E2 3324.843} C_VEL
LIN {X 0,Y 553.177,Z 360.379,A -85,B 0,C 180,E1 3326.677,E2 3326.677} C_VEL
LIN {X 0,Y 552.884,Z 376.9,A -85,B 0,C 180,E1 3329.023,E2 3329.023} C_VEL
LIN {X 0,Y 552.693,Z 387.926,A -85,B 0,C 180,E1 3331.565,E2 3331.565} C_VEL
LIN {X 0,Y 552.731,Z 393.482,A -85,B 0,C 180,E1 3333.914,E2 3333.914} C_VEL
LIN {X 0,Y 552.561,Z 394.939,A -85,B 0,C 180,E1 3336.272,E2 3336.272} C_VEL
LIN {X 0,Y 552.633,Z 392.38,A -85,B 0,C 180,E1 3338.638,E2 3338.638} C_VEL
LIN {X 0,Y 552.719,Z 383.992,A -85,B 0,C 180,E1 3341.417,E2 3341.417} C_VEL
LIN {X 0,Y 552.932,Z 371.252,A -85,B 0,C 180,E1 3343.816,E2 3343.816} C_VEL
LIN {X 0,Y 553.282,Z 352.779,A -85,B 0,C 180,E1 3346.031,E2 3346.031} C_VEL
LIN {X 0,Y 553.809,Z 330.476,A -85,B 0,C 180,E1 3347.749,E2 3347.749} C_VEL
LIN {X 0,Y 553.728,Z 305.215,A -85,B 0,C 180,E1 3348.937,E2 3348.937} C_VEL
LIN {X 0,Y 552.445,Z 297.81,A -85,B 0,C 180,E1 3349.269,E2 3349.269} C_VEL
LIN {X 0,Y 551.994,Z 297.81,A -85,B 0,C 180,E1 3355.938,E2 3355.938} C_VEL
LIN {X 0,Y 551.842,Z 297.81,A -85,B 0,C 180,E1 3362.018,E2 3362.018} C_VEL
LIN {X 0,Y 552.066,Z 297.81,A -85,B 0,C 180,E1 3367.545,E2 3367.545} C_VEL
LIN {X 0,Y 551.831,Z 297.81,A -85,B 0,C 180,E1 3373.129,E2 3373.129} C_VEL
LIN {X 0,Y 551.977,Z 297.81,A -85,B 0,C 180,E1 3378.981,E2 3378.981} C_VEL
LIN {X 0,Y 551.943,Z 297.81,A -85,B 0,C 180,E1 3384.948,E2 3384.948} C_VEL
LIN {X 0,Y 551.942,Z 297.81,A -85,B 0,C 180,E1 3391.031,E2 3391.031} C_VEL
LIN {X 0,Y 551.977,Z 297.81,A -85,B 0,C 180,E1 3395.779,E2 3395.779} C_VEL
LIN {X 0,Y 552.278,Z 297.81,A -85,B 0,C 180,E1 3400.849,E2 3400.849} C_VEL
LIN {X 0,Y 551.955,Z 297.81,A -85,B 0,C 180,E1 3405.745,E2 3405.745} C_VEL
LIN {X 0,Y 552.183,Z 297.81,A -85,B 0,C 180,E1 3410.553,E2 3410.553} C_VEL
LIN {X 0,Y 552.274,Z 297.81,A -85,B 0,C 180,E1 3415.288,E2 3415.288} C_VEL
LIN {X 0,Y 552.358,Z 297.81,A -85,B 0,C 180,E1 3419.99,E2 3419.99} C_VEL
LIN {X 0,Y 552.347,Z 297.81,A -85,B 0,C 180,E1 3424.692,E2 3424.692} C_VEL
LIN {X 0,Y 552.158,Z 297.81,A -85,B 0,C 180,E1 3430.31,E2 3430.31} C_VEL
LIN {X 0,Y 552.078,Z 297.81,A -85,B 0,C 180,E1 3436.137,E2 3436.137} C_VEL
LIN {X 0,Y 552.1,Z 297.81,A -85,B 0,C 180,E1 3439.651,E2 3439.651} C_VEL
LIN {X 0,Y 548.101,Z 297.81,A -85,B 0,C 180,E1 3441.42,E2 3441.42} C_VEL
LIN {X 0,Y 544.11,Z 297.81,A -85,B 0,C 180,E1 3443.214,E2 3443.214} C_VEL
LIN {X 0,Y 544.089,Z 297.81,A -85,B 0,C 180,E1 3448.12,E2 3448.12} C_VEL
LIN {X 0,Y 544.055,Z 297.81,A -85,B 0,C 180,E1 3453.686,E2 3453.686} C_VEL
LIN {X 0,Y 543.922,Z 297.81,A -85,B 0,C 180,E1 3459.638,E2 3459.638} C_VEL
LIN {X 0,Y 544.021,Z 297.81,A -85,B 0,C 180,E1 3466.14,E2 3466.14} C_VEL
LIN {X 0,Y 544.101,Z 297.81,A -85,B 0,C 180,E1 3472.4,E2 3472.4} C_VEL
LIN {X 0,Y 544.05,Z 297.81,A -85,B 0,C 180,E1 3478.197,E2 3478.197} C_VEL
LIN {X 0,Y 544.153,Z 297.81,A -85,B 0,C 180,E1 3483.659,E2 3483.659} C_VEL
LIN {X 0,Y 544.492,Z 297.81,A -85,B 0,C 180,E1 3486.508,E2 3486.508} C_VEL
LIN {X 0,Y 549.188,Z 314.803,A -85,B 0,C 180,E1 3486.918,E2 3486.918} C_VEL
LIN {X 0,Y 548.979,Z 376.881,A -85,B 0,C 180,E1 3487.845,E2 3487.845} C_VEL
LIN {X 0,Y 548.289,Z 410.061,A -85,B 0,C 180,E1 3488.934,E2 3488.934} C_VEL
LIN {X 0,Y 547.431,Z 442.932,A -85,B 0,C 180,E1 3490.683,E2 3490.683} C_VEL
LIN {X 0,Y 546.567,Z 472.126,A -85,B 0,C 180,E1 3492.941,E2 3492.941} C_VEL
LIN {X 0,Y 545.71,Z 496.037,A -85,B 0,C 180,E1 3495.589,E2 3495.589} C_VEL
LIN {X 0,Y 545.147,Z 515.826,A -85,B 0,C 180,E1 3498.625,E2 3498.625} C_VEL
LIN {X 0,Y 544.871,Z 531.183,A -85,B 0,C 180,E1 3502.04,E2 3502.04} C_VEL
LIN {X 0,Y 544.719,Z 540.948,A -85,B 0,C 180,E1 3505.666,E2 3505.666} C_VEL
LIN {X 0,Y 544.682,Z 544.419,A -85,B 0,C 180,E1 3508.412,E2 3508.412} C_VEL
LIN {X 0,Y 544.64,Z 544.419,A -85,B 0,C 180,E1 3511.587,E2 3511.587} C_VEL
LIN {X 0,Y 544.711,Z 540.1,A -85,B 0,C 180,E1 3514.767,E2 3514.767} C_VEL
LIN {X 0,Y 544.888,Z 529.67,A -85,B 0,C 180,E1 3518.36,E2 3518.36} C_VEL
LIN {X 0,Y 545.223,Z 513.596,A -85,B 0,C 180,E1 3521.777,E2 3521.777} C_VEL
LIN {X 0,Y 545.843,Z 492.459,A -85,B 0,C 180,E1 3524.867,E2 3524.867} C_VEL
LIN {X 0,Y 546.643,Z 467.542,A -85,B 0,C 180,E1 3527.469,E2 3527.469} C_VEL
LIN {X 0,Y 547.548,Z 437.847,A -85,B 0,C 180,E1 3529.634,E2 3529.634} C_VEL
LIN {X 0,Y 548.396,Z 405.049,A -85,B 0,C 180,E1 3531.262,E2 3531.262} C_VEL
LIN {X 0,Y 548.945,Z 371.842,A -85,B 0,C 180,E1 3532.253,E2 3532.253} C_VEL
LIN {X 0,Y 548.417,Z 311.557,A -85,B 0,C 180,E1 3533.133,E2 3533.133} C_VEL
LIN {X 0,Y 544.361,Z 297.81,A -85,B 0,C 180,E1 3533.53,E2 3533.53} C_VEL
LIN {X 0,Y 544.015,Z 297.81,A -85,B 0,C 180,E1 3539.952,E2 3539.952} C_VEL
LIN {X 0,Y 543.918,Z 297.81,A -85,B 0,C 180,E1 3545.633,E2 3545.633} C_VEL
LIN {X 0,Y 543.889,Z 297.81,A -85,B 0,C 180,E1 3551.748,E2 3551.748} C_VEL
LIN {X 0,Y 544.013,Z 297.81,A -85,B 0,C 180,E1 3558.274,E2 3558.274} C_VEL
LIN {X 0,Y 543.953,Z 297.81,A -85,B 0,C 180,E1 3564.38,E2 3564.38} C_VEL
LIN {X 0,Y 543.968,Z 297.81,A -85,B 0,C 180,E1 3570.055,E2 3570.055} C_VEL
LIN {X 0,Y 544.082,Z 297.81,A -85,B 0,C 180,E1 3575.426,E2 3575.426} C_VEL
LIN {X 0,Y 544.242,Z 297.81,A -85,B 0,C 180,E1 3580.576,E2 3580.576} C_VEL
LIN {X 0,Y 543.952,Z 297.81,A -85,B 0,C 180,E1 3586.153,E2 3586.153} C_VEL
LIN {X 0,Y 544.239,Z 297.81,A -85,B 0,C 180,E1 3590.433,E2 3590.433} C_VEL
LIN {X 0,Y 544.418,Z 297.81,A -85,B 0,C 180,E1 3595.24,E2 3595.24} C_VEL
LIN {X 0,Y 544.412,Z 297.81,A -85,B 0,C 180,E1 3600.01,E2 3600.01} C_VEL
LIN {X 0,Y 544.348,Z 297.81,A -85,B 0,C 180,E1 3604.781,E2 3604.781} C_VEL
LIN {X 0,Y 544.347,Z 297.81,A -85,B 0,C 180,E1 3609.585,E2 3609.585} C_VEL
LIN {X 0,Y 544.289,Z 297.81,A -85,B 0,C 180,E1 3614.46,E2 3614.46} C_VEL
LIN {X 0,Y 544.232,Z 297.81,A -85,B 0,C 180,E1 3619.488,E2 3619.488} C_VEL
LIN {X 0,Y 544.088,Z 297.81,A -85,B 0,C 180,E1 3624.595,E2 3624.595} C_VEL
LIN {X 0,Y 544.052,Z 297.81,A -85,B 0,C 180,E1 3630.704,E2 3630.704} C_VEL
LIN {X 0,Y 544.387,Z 298.529,A -85,B 0,C 180,E1 3636.387,E2 3636.387} C_VEL
LIN {X 0,Y 546.594,Z 312.917,A -85,B 0,C 180,E1 3636.97,E2 3636.97} C_VEL
LIN {X 0,Y 546.158,Z 337.855,A -85,B 0,C 180,E1 3638.356,E2 3638.356} C_VEL
LIN {X 0,Y 545.582,Z 359.886,A -85,B 0,C 180,E1 3640.33,E2 3640.33} C_VEL
LIN {X 0,Y 545.126,Z 376.678,A -85,B 0,C 180,E1 3642.666,E2 3642.666} C_VEL
LIN {X 0,Y 544.939,Z 388.391,A -85,B 0,C 180,E1 3645.298,E2 3645.298} C_VEL
LIN {X 0,Y 544.772,Z 393.985,A -85,B 0,C 180,E1 3647.58,E2 3647.58} C_VEL
LIN {X 0,Y 544.637,Z 395.568,A -85,B 0,C 180,E1 3650.894,E2 3650.894} C_VEL
LIN {X 0,Y 544.813,Z 391.641,A -85,B 0,C 180,E1 3653.459,E2 3653.459} C_VEL
LIN {X 0,Y 545.011,Z 382.036,A -85,B 0,C 180,E1 3656.183,E2 3656.183} C_VEL
LIN {X 0,Y 545.347,Z 366.662,A -85,B 0,C 180,E1 3658.728,E2 3658.728} C_VEL
LIN {X 0,Y 545.824,Z 347.143,A -85,B 0,C 180,E1 3660.799,E2 3660.799} C_VEL
LIN {X 0,Y 546.322,Z 323.347,A -85,B 0,C 180,E1 3662.418,E2 3662.418} C_VEL
LIN {X 0,Y 545.497,Z 302.547,A -85,B 0,C 180,E1 3663.327,E2 3663.327} C_VEL
LIN {X 0,Y 544.56,Z 297.81,A -85,B 0,C 180,E1 3663.581,E2 3663.581} C_VEL
LIN {X 0,Y 544.29,Z 297.81,A -85,B 0,C 180,E1 3670.568,E2 3670.568} C_VEL
LIN {X 0,Y 543.997,Z 297.81,A -85,B 0,C 180,E1 3676.185,E2 3676.185} C_VEL
LIN {X 0,Y 544.319,Z 297.81,A -85,B 0,C 180,E1 3682.033,E2 3682.033} C_VEL
LIN {X 0,Y 544.423,Z 297.835,A -85,B 0,C 180,E1 3682.485,E2 3682.485} C_VEL
LIN {X 0,Y 546.389,Z 315.548,A -85,B 0,C 180,E1 3683.16,E2 3683.16} C_VEL
LIN {X 0,Y 545.983,Z 340.11,A -85,B 0,C 180,E1 3684.573,E2 3684.573} C_VEL
LIN {X 0,Y 545.476,Z 360.432,A -85,B 0,C 180,E1 3686.432,E2 3686.432} C_VEL
LIN {X 0,Y 545.126,Z 377.322,A -85,B 0,C 180,E1 3688.811,E2 3688.811} C_VEL
LIN {X 0,Y 544.879,Z 387.981,A -85,B 0,C 180,E1 3691.191,E2 3691.191} C_VEL
LIN {X 0,Y 544.866,Z 393.199,A -85,B 0,C 180,E1 3693.176,E2 3693.176} C_VEL
LIN {X 0,Y 544.806,Z 395.378,A -85,B 0,C 180,E1 3694.767,E2 3694.767} C_VEL
LIN {X 0,Y 544.717,Z 395.792,A -85,B 0,C 180,E1 3696.362,E2 3696.362} C_VEL
LIN {X 0,Y 544.807,Z 393.159,A -85,B 0,C 180,E1 3698.763,E2 3698.763} C_VEL
LIN {X 0,Y 544.95,Z 384.714,A -85,B 0,C 180,E1 3701.582,E2 3701.582} C_VEL
LIN {X 0,Y 545.232,Z 370.723,A -85,B 0,C 180,E1 3704.164,E2 3704.164} C_VEL
LIN {X 0,Y 545.624,Z 353.191,A -85,B 0,C 180,E1 3706.24,E2 3706.24} C_VEL
LIN {X 0,Y 546.191,Z 330.129,A -85,B 0,C 180,E1 3708.005,E2 3708.005} C_VEL
LIN {X 0,Y 545.892,Z 305.195,A -85,B 0,C 180,E1 3709.164,E2 3709.164} C_VEL
LIN {X 0,Y 544.521,Z 297.81,A -85,B 0,C 180,E1 3709.494,E2 3709.494} C_VEL
LIN {X 0,Y 544.021,Z 297.81,A -85,B 0,C 180,E1 3716.347,E2 3716.347} C_VEL
LIN {X 0,Y 543.947,Z 297.81,A -85,B 0,C 180,E1 3721.81,E2 3721.81} C_VEL
LIN {X 0,Y 544.177,Z 297.81,A -85,B 0,C 180,E1 3727.594,E2 3727.594} C_VEL
LIN {X 0,Y 543.915,Z 297.81,A -85,B 0,C 180,E1 3733.915,E2 3733.915} C_VEL
LIN {X 0,Y 544.04,Z 297.81,A -85,B 0,C 180,E1 3738.495,E2 3738.495} C_VEL
LIN {X 0,Y 543.989,Z 297.81,A -85,B 0,C 180,E1 3744.358,E2 3744.358} C_VEL
LIN {X 0,Y 543.975,Z 297.81,A -85,B 0,C 180,E1 3750.032,E2 3750.032} C_VEL
LIN {X 0,Y 544.069,Z 297.81,A -85,B 0,C 180,E1 3756.245,E2 3756.245} C_VEL
LIN {X 0,Y 544.369,Z 297.81,A -85,B 0,C 180,E1 3762.236,E2 3762.236} C_VEL
LIN {X 0,Y 544.269,Z 297.81,A -85,B 0,C 180,E1 3768.799,E2 3768.799} C_VEL
LIN {X 0,Y 544.524,Z 297.81,A -85,B 0,C 180,E1 3773.626,E2 3773.626} C_VEL
LIN {X 0,Y 544.456,Z 297.81,A -85,B 0,C 180,E1 3779.99,E2 3779.99} C_VEL
LIN {X 0,Y 544.441,Z 297.81,A -85,B 0,C 180,E1 3784.76,E2 3784.76} C_VEL
LIN {X 0,Y 544.366,Z 297.81,A -85,B 0,C 180,E1 3789.564,E2 3789.564} C_VEL
LIN {X 0,Y 544.336,Z 297.81,A -85,B 0,C 180,E1 3794.438,E2 3794.438} C_VEL
LIN {X 0,Y 544.212,Z 297.81,A -85,B 0,C 180,E1 3799.64,E2 3799.64} C_VEL
LIN {X 0,Y 544.11,Z 297.81,A -85,B 0,C 180,E1 3803.214,E2 3803.214} C_VEL
LIN {X 0,Y 540.153,Z 297.81,A -85,B 0,C 180,E1 3805.016,E2 3805.016} C_VEL
LIN {X 0,Y 536.116,Z 297.81,A -85,B 0,C 180,E1 3806.844,E2 3806.844} C_VEL
LIN {X 0,Y 536.123,Z 297.81,A -85,B 0,C 180,E1 3812.392,E2 3812.392} C_VEL
LIN {X 0,Y 536.027,Z 297.81,A -85,B 0,C 180,E1 3818.256,E2 3818.256} C_VEL
LIN {X 0,Y 535.994,Z 297.81,A -85,B 0,C 180,E1 3824.723,E2 3824.723} C_VEL
LIN {X 0,Y 536.099,Z 297.81,A -85,B 0,C 180,E1 3829.654,E2 3829.654} C_VEL
LIN {X 0,Y 536.045,Z 297.81,A -85,B 0,C 180,E1 3835.735,E2 3835.735} C_VEL
LIN {X 0,Y 536.129,Z 297.81,A -85,B 0,C 180,E1 3841.413,E2 3841.413} C_VEL
LIN {X 0,Y 536.561,Z 297.81,A -85,B 0,C 180,E1 3846.215,E2 3846.215} C_VEL
LIN {X 0,Y 541.701,Z 317.008,A -85,B 0,C 180,E1 3846.682,E2 3846.682} C_VEL
LIN {X 0,Y 541.429,Z 377.357,A -85,B 0,C 180,E1 3847.608,E2 3847.608} C_VEL
LIN {X 0,Y 540.661,Z 410.47,A -85,B 0,C 180,E1 3848.725,E2 3848.725} C_VEL
LIN {X 0,Y 539.693,Z 442.973,A -85,B 0,C 180,E1 3850.501,E2 3850.501} C_VEL
LIN {X 0,Y 538.727,Z 472.461,A -85,B 0,C 180,E1 3852.839,E2 3852.839} C_VEL
LIN {X 0,Y 537.91,Z 497.42,A -85,B 0,C 180,E1 3855.583,E2 3855.583} C_VEL
LIN {X 0,Y 537.282,Z 516.907,A -85,B 0,C 180,E1 3858.661,E2 3858.661} C_VEL
LIN {X 0,Y 536.98,Z 531.183,A -85,B 0,C 180,E1 3861.922,E2 3861.922} C_VEL
LIN {X 0,Y 536.828,Z 540.097,A -85,B 0,C 180,E1 3865.162,E2 3865.162} C_VEL
LIN {X 0,Y 536.806,Z 544.419,A -85,B 0,C 180,E1 3868.389,E2 3868.389} C_VEL
LIN {X 0,Y 536.766,Z 544.419,A -85,B 0,C 180,E1 3871.61,E2 3871.61} C_VEL
LIN {X 0,Y 536.813,Z 540.099,A -85,B 0,C 180,E1 3874.837,E2 3874.837} C_VEL
LIN {X 0,Y 536.998,Z 529.67,A -85,B 0,C 180,E1 3878.483,E2 3878.483} C_VEL
LIN {X 0,Y 537.394,Z 513.595,A -85,B 0,C 180,E1 3881.951,E2 3881.951} C_VEL
LIN {X 0,Y 538.023,Z 493.779,A -85,B 0,C 180,E1 3884.869,E2 3884.869} C_VEL
LIN {X 0,Y 538.856,Z 467.544,A -85,B 0,C 180,E1 3887.6,E2 3887.6} C_VEL
LIN {X 0,Y 539.828,Z 437.879,A -85,B 0,C 180,E1 3889.817,E2 3889.817} C_VEL
LIN {X 0,Y 540.761,Z 405.015,A -85,B 0,C 180,E1 3891.484,E2 3891.484} C_VEL
LIN {X 0,Y 541.432,Z 370.937,A -85,B 0,C 180,E1 3892.517,E2 3892.517} C_VEL
LIN {X 0,Y 540.86,Z 313.269,A -85,B 0,C 180,E1 3893.372,E2 3893.372} C_VEL
LIN {X 0,Y 536.417,Z 297.81,A -85,B 0,C 180,E1 3893.786,E2 3893.786} C_VEL
LIN {X 0,Y 536.124,Z 297.81,A -85,B 0,C 180,E1 3900.439,E2 3900.439} C_VEL
LIN {X 0,Y 535.991,Z 297.81,A -85,B 0,C 180,E1 3906.243,E2 3906.243} C_VEL
LIN {X 0,Y 535.904,Z 297.81,A -85,B 0,C 180,E1 3912.515,E2 3912.515} C_VEL
LIN {X 0,Y 536.009,Z 297.81,A -85,B 0,C 180,E1 3917.507,E2 3917.507} C_VEL
LIN {X 0,Y 536.066,Z 297.81,A -85,B 0,C 180,E1 3923.773,E2 3923.773} C_VEL
LIN {X 0,Y 536.058,Z 297.81,A -85,B 0,C 180,E1 3929.566,E2 3929.566} C_VEL
LIN {X 0,Y 536.135,Z 297.81,A -85,B 0,C 180,E1 3935.037,E2 3935.037} C_VEL
LIN {X 0,Y 536.312,Z 297.81,A -85,B 0,C 180,E1 3940.277,E2 3940.277} C_VEL
LIN {X 0,Y 536.089,Z 297.81,A -85,B 0,C 180,E1 3945.335,E2 3945.335} C_VEL
LIN {X 0,Y 536.319,Z 297.81,A -85,B 0,C 180,E1 3950.291,E2 3950.291} C_VEL
LIN {X 0,Y 536.514,Z 297.81,A -85,B 0,C 180,E1 3955.17,E2 3955.17} C_VEL
LIN {X 0,Y 536.519,Z 297.81,A -85,B 0,C 180,E1 3960.01,E2 3960.01} C_VEL
LIN {X 0,Y 536.438,Z 297.81,A -85,B 0,C 180,E1 3964.851,E2 3964.851} C_VEL
LIN {X 0,Y 536.371,Z 297.81,A -85,B 0,C 180,E1 3970.048,E2 3970.048} C_VEL
LIN {X 0,Y 536.353,Z 297.81,A -85,B 0,C 180,E1 3974.678,E2 3974.678} C_VEL
LIN {X 0,Y 536.314,Z 297.81,A -85,B 0,C 180,E1 3979.744,E2 3979.744} C_VEL
LIN {X 0,Y 536.094,Z 297.81,A -85,B 0,C 180,E1 3985.746,E2 3985.746} C_VEL
LIN {X 0,Y 536.141,Z 297.81,A -85,B 0,C 180,E1 3990.452,E2 3990.452} C_VEL
LIN {X 0,Y 536.428,Z 297.892,A -85,B 0,C 180,E1 3996.089,E2 3996.089} C_VEL
LIN {X 0,Y 539.058,Z 314.04,A -85,B 0,C 180,E1 3996.753,E2 3996.753} C_VEL
LIN {X 0,Y 538.585,Z 338.561,A -85,B 0,C 180,E1 3998.137,E2 3998.137} C_VEL
LIN {X 0,Y 537.958,Z 360.134,A -85,B 0,C 180,E1 4000.08,E2 4000.08} C_VEL
LIN {X 0,Y 537.402,Z 376.852,A -85,B 0,C 180,E1 4002.385,E2 4002.385} C_VEL
LIN {X 0,Y 537.171,Z 388.816,A -85,B 0,C 180,E1 4005.008,E2 4005.008} C_VEL
LIN {X 0,Y 536.953,Z 395.163,A -85,B 0,C 180,E1 4007.588,E2 4007.588} C_VEL
LIN {X 0,Y 536.797,Z 396.966,A -85,B 0,C 180,E1 4009.718,E2 4009.718} C_VEL
LIN {X 0,Y 536.963,Z 394.175,A -85,B 0,C 180,E1 4012.835,E2 4012.835} C_VEL
LIN {X 0,Y 537.202,Z 385.935,A -85,B 0,C 180,E1 4015.624,E2 4015.624} C_VEL
LIN {X 0,Y 537.512,Z 372.254,A -85,B 0,C 180,E1 4018.219,E2 4018.219} C_VEL
LIN {X 0,Y 538.012,Z 354.035,A -85,B 0,C 180,E1 4020.421,E2 4020.421} C_VEL
LIN {X 0,Y 538.6,Z 332.637,A -85,B 0,C 180,E1 4022.13,E2 4022.13} C_VEL
LIN {X 0,Y 538.509,Z 306.341,A -85,B 0,C 180,E1 4023.432,E2 4023.432} C_VEL
LIN {X 0,Y 536.583,Z 297.81,A -85,B 0,C 180,E1 4023.817,E2 4023.817} C_VEL
LIN {X 0,Y 536.387,Z 297.81,A -85,B 0,C 180,E1 4030.27,E2 4030.27} C_VEL
LIN {X 0,Y 536.124,Z 297.81,A -85,B 0,C 180,E1 4035.327,E2 4035.327} C_VEL
LIN {X 0,Y 536.382,Z 297.81,A -85,B 0,C 180,E1 4040.283,E2 4040.283} C_VEL
LIN {X 0,Y 536.5,Z 298.446,A -85,B 0,C 180,E1 4042.272,E2 4042.272} C_VEL
LIN {X 0,Y 538.771,Z 316.268,A -85,B 0,C 180,E1 4042.962,E2 4042.962} C_VEL
LIN {X 0,Y 538.343,Z 340.54,A -85,B 0,C 180,E1 4044.363,E2 4044.363} C_VEL
LIN {X 0,Y 537.753,Z 362.256,A -85,B 0,C 180,E1 4046.381,E2 4046.381} C_VEL
LIN {X 0,Y 537.381,Z 378.871,A -85,B 0,C 180,E1 4048.794,E2 4048.794} C_VEL
LIN {X 0,Y 537.122,Z 390.586,A -85,B 0,C 180,E1 4051.61,E2 4051.61} C_VEL
LIN {X 0,Y 537.023,Z 396.024,A -85,B 0,C 180,E1 4054.316,E2 4054.316} C_VEL
LIN {X 0,Y 536.893,Z 396.855,A -85,B 0,C 180,E1 4056.456,E2 4056.456} C_VEL
LIN {X 0,Y 537.028,Z 394.076,A -85,B 0,C 180,E1 4058.891,E2 4058.891} C_VEL
LIN {X 0,Y 537.186,Z 385.436,A -85,B 0,C 180,E1 4061.751,E2 4061.751} C_VEL
LIN {X 0,Y 537.515,Z 371.196,A -85,B 0,C 180,E1 4064.372,E2 4064.372} C_VEL
LIN {X 0,Y 537.951,Z 353.577,A -85,B 0,C 180,E1 4066.454,E2 4066.454} C_VEL
LIN {X 0,Y 538.537,Z 331.432,A -85,B 0,C 180,E1 4068.164,E2 4068.164} C_VEL
LIN {X 0,Y 538.182,Z 305.896,A -85,B 0,C 180,E1 4069.369,E2 4069.369} C_VEL
LIN {X 0,Y 536.559,Z 297.81,A -85,B 0,C 180,E1 4069.724,E2 4069.724} C_VEL
LIN {X 0,Y 536.087,Z 297.81,A -85,B 0,C 180,E1 4075.717,E2 4075.717} C_VEL
LIN {X 0,Y 536.069,Z 297.81,A -85,B 0,C 180,E1 4080.444,E2 4080.444} C_VEL
LIN {X 0,Y 536.17,Z 297.81,A -85,B 0,C 180,E1 4086.23,E2 4086.23} C_VEL
LIN {X 0,Y 536.04,Z 297.81,A -85,B 0,C 180,E1 4090.512,E2 4090.512} C_VEL
LIN {X 0,Y 536.027,Z 297.81,A -85,B 0,C 180,E1 4097.05,E2 4097.05} C_VEL
LIN {X 0,Y 536.156,Z 297.81,A -85,B 0,C 180,E1 4102.005,E2 4102.005} C_VEL
LIN {X 0,Y 536.013,Z 297.81,A -85,B 0,C 180,E1 4107.65,E2 4107.65} C_VEL
LIN {X 0,Y 536.091,Z 297.81,A -85,B 0,C 180,E1 4113.22,E2 4113.22} C_VEL
LIN {X 0,Y 536.27,Z 297.81,A -85,B 0,C 180,E1 4118.531,E2 4118.531} C_VEL
LIN {X 0,Y 536.333,Z 297.81,A -85,B 0,C 180,E1 4123.648,E2 4123.648} C_VEL
LIN {X 0,Y 536.379,Z 297.81,A -85,B 0,C 180,E1 4130.272,E2 4130.272} C_VEL
LIN {X 0,Y 536.474,Z 297.81,A -85,B 0,C 180,E1 4135.149,E2 4135.149} C_VEL
LIN {X 0,Y 536.586,Z 297.81,A -85,B 0,C 180,E1 4139.99,E2 4139.99} C_VEL
LIN {X 0,Y 536.526,Z 297.81,A -85,B 0,C 180,E1 4144.83,E2 4144.83} C_VEL
LIN {X 0,Y 536.413,Z 297.81,A -85,B 0,C 180,E1 4150.068,E2 4150.068} C_VEL
LIN {X 0,Y 536.391,Z 297.81,A -85,B 0,C 180,E1 4154.657,E2 4154.657} C_VEL
LIN {X 0,Y 536.325,Z 297.81,A -85,B 0,C 180,E1 4159.723,E2 4159.723} C_VEL
LIN {X 0,Y 536.093,Z 297.81,A -85,B 0,C 180,E1 4165.744,E2 4165.744} C_VEL
LIN {X 0,Y 536.116,Z 297.81,A -85,B 0,C 180,E1 4166.844,E2 4166.844} C_VEL
LIN {X 0,Y 532.033,Z 297.81,A -85,B 0,C 180,E1 4168.674,E2 4168.674} C_VEL
LIN {X 0,Y 528.113,Z 297.81,A -85,B 0,C 180,E1 4170.531,E2 4170.531} C_VEL
LIN {X 0,Y 528.122,Z 297.81,A -85,B 0,C 180,E1 4174.841,E2 4174.841} C_VEL
LIN {X 0,Y 528.003,Z 297.81,A -85,B 0,C 180,E1 4181.084,E2 4181.084} C_VEL
LIN {X 0,Y 528.11,Z 297.81,A -85,B 0,C 180,E1 4186.704,E2 4186.704} C_VEL
LIN {X 0,Y 528.187,Z 297.81,A -85,B 0,C 180,E1 4193.11,E2 4193.11} C_VEL
LIN {X 0,Y 528.178,Z 297.81,A -85,B 0,C 180,E1 4199.052,E2 4199.052} C_VEL
LIN {X 0,Y 528.611,Z 297.81,A -85,B 0,C 180,E1 4205.91,E2 4205.91} C_VEL
LIN {X 0,Y 534.25,Z 319.391,A -85,B 0,C 180,E1 4206.441,E2 4206.441} C_VEL
LIN {X 0,Y 533.91,Z 377.186,A -85,B 0,C 180,E1 4207.347,E2 4207.347} C_VEL
LIN {X 0,Y 533.049,Z 411.38,A -85,B 0,C 180,E1 4208.533,E2 4208.533} C_VEL
LIN {X 0,Y 531.972,Z 443.015,A -85,B 0,C 180,E1 4210.315,E2 4210.315} C_VEL
LIN {X 0,Y 530.91,Z 470.979,A -85,B 0,C 180,E1 4212.565,E2 4212.565} C_VEL
LIN {X 0,Y 530.034,Z 496.665,A -85,B 0,C 180,E1 4215.427,E2 4215.427} C_VEL
LIN {X 0,Y 529.386,Z 517.465,A -85,B 0,C 180,E1 4218.683,E2 4218.683} C_VEL
LIN {X 0,Y 529.089,Z 531.18,A -85,B 0,C 180,E1 4221.801,E2 4221.801} C_VEL
LIN {X 0,Y 528.927,Z 540.096,A -85,B 0,C 180,E1 4225.09,E2 4225.09} C_VEL
LIN {X 0,Y 528.902,Z 544.418,A -85,B 0,C 180,E1 4228.365,E2 4228.365} C_VEL
LIN {X 0,Y 528.863,Z 544.418,A -85,B 0,C 180,E1 4231.635,E2 4231.635} C_VEL
LIN {X 0,Y 528.915,Z 540.098,A -85,B 0,C 180,E1 4234.909,E2 4234.909} C_VEL
LIN {X 0,Y 529.126,Z 529.655,A -85,B 0,C 180,E1 4238.61,E2 4238.61} C_VEL
LIN {X 0,Y 529.523,Z 514.14,A -85,B 0,C 180,E1 4241.923,E2 4241.923} C_VEL
LIN {X 0,Y 530.172,Z 492.771,A -85,B 0,C 180,E1 4245.053,E2 4245.053} C_VEL
LIN {X 0,Y 531.081,Z 466.572,A -85,B 0,C 180,E1 4247.82,E2 4247.82} C_VEL
LIN {X 0,Y 532.111,Z 437.82,A -85,B 0,C 180,E1 4250.007,E2 4250.007} C_VEL
LIN {X 0,Y 533.154,Z 404.739,A -85,B 0,C 180,E1 4251.723,E2 4251.723} C_VEL
LIN {X 0,Y 533.919,Z 371.097,A -85,B 0,C 180,E1 4252.768,E2 4252.768} C_VEL
LIN {X 0,Y 533.322,Z 314.761,A -85,B 0,C 180,E1 4253.623,E2 4253.623} C_VEL
LIN {X 0,Y 528.439,Z 297.81,A -85,B 0,C 180,E1 4254.102,E2 4254.102} C_VEL
LIN {X 0,Y 528.226,Z 297.81,A -85,B 0,C 180,E1 4259.054,E2 4259.054} C_VEL
LIN {X 0,Y 528.134,Z 297.81,A -85,B 0,C 180,E1 4264.85,E2 4264.85} C_VEL
LIN {X 0,Y 527.949,Z 297.81,A -85,B 0,C 180,E1 4271.101,E2 4271.101} C_VEL
LIN {X 0,Y 528.042,Z 297.81,A -85,B 0,C 180,E1 4276.71,E2 4276.71} C_VEL
LIN {X 0,Y 528.144,Z 297.81,A -85,B 0,C 180,E1 4283.13,E2 4283.13} C_VEL
LIN {X 0,Y 528.113,Z 297.81,A -85,B 0,C 180,E1 4289.059,E2 4289.059} C_VEL
LIN {X 0,Y 528.226,Z 297.81,A -85,B 0,C 180,E1 4294.637,E2 4294.637} C_VEL
LIN {X 0,Y 528.41,Z 297.81,A -85,B 0,C 180,E1 4300.455,E2 4300.455} C_VEL
LIN {X 0,Y 528.15,Z 297.81,A -85,B 0,C 180,E1 4306.268,E2 4306.268} C_VEL
LIN {X 0,Y 528.408,Z 297.81,A -85,B 0,C 180,E1 4311.801,E2 4311.801} C_VEL
LIN {X 0,Y 528.639,Z 297.81,A -85,B 0,C 180,E1 4317.52,E2 4317.52} C_VEL
LIN {X 0,Y 528.675,Z 297.81,A -85,B 0,C 180,E1 4323.283,E2 4323.283} C_VEL
LIN {X 0,Y 528.559,Z 297.81,A -85,B 0,C 180,E1 4328.217,E2 4328.217} C_VEL
LIN {X 0,Y 528.431,Z 297.81,A -85,B 0,C 180,E1 4333.856,E2 4333.856} C_VEL
LIN {X 0,Y 528.381,Z 297.81,A -85,B 0,C 180,E1 4340.053,E2 4340.053} C_VEL
LIN {X 0,Y 528.217,Z 297.81,A -85,B 0,C 180,E1 4345.386,E2 4345.386} C_VEL
LIN {X 0,Y 528.195,Z 297.81,A -85,B 0,C 180,E1 4351.012,E2 4351.012} C_VEL
LIN {X 0,Y 528.504,Z 297.81,A -85,B 0,C 180,E1 4355.786,E2 4355.786} C_VEL
LIN {X 0,Y 531.503,Z 315.732,A -85,B 0,C 180,E1 4356.555,E2 4356.555} C_VEL
LIN {X 0,Y 530.961,Z 339.997,A -85,B 0,C 180,E1 4357.966,E2 4357.966} C_VEL
LIN {X 0,Y 530.282,Z 361.953,A -85,B 0,C 180,E1 4359.998,E2 4359.998} C_VEL
LIN {X 0,Y 529.659,Z 378.639,A -85,B 0,C 180,E1 4362.38,E2 4362.38} C_VEL
LIN {X 0,Y 529.373,Z 390.334,A -85,B 0,C 180,E1 4365.054,E2 4365.054} C_VEL
LIN {X 0,Y 529.125,Z 396.735,A -85,B 0,C 180,E1 4367.875,E2 4367.875} C_VEL
